FUNCTION "Op20.FCCycles" : VOID	// FC 170
VERSION : 0.1
BEGIN
NETWORK
TITLE =
      A     "OP20".Mode.Automatic;
      FP    "AppoFP_M51.6";
      =     "Op20.Bench.Systems".State.FP_Mode_automatic;
      AN    "OP20".Diagnostic.Alarm_Stop_Cycle;
      AN    "OP20".Diagnostic.Alarm_Emergency;
      FP    "AppoFP_M51.7";
      =     "Op20.Bench.Systems".State.FP_uscita_da_allarme;
NETWORK
TITLE = Attiva ciclo
      A     "Op20.Bench.Systems".State.FP_Mode_automatic;
      O     "Op20.Bench.Systems".State.FP_uscita_da_allarme;
      A(;
      AN    "Op20.Bench.MapE".Index_cassetto_Giu;
      ON    "Op20.Bench.MapE".Gruppo_piantaggio_Su;
      ON    "Op20.Bench.MapE".Piantaggio_Su;
      );
      S     "Op20.Cycles".Restore.Command.Activate_Cycle;
      AN    "OP20".Mode.Automatic;
      O     "OP20".Diagnostic.Alarm_Stop_Cycle;
      O     "OP20".Diagnostic.Alarm_Emergency;
      O     "Op20.Cycles".Restore.State.State_Bit[60];
      R     "Op20.Cycles".Restore.Command.Activate_Cycle;
      CLR;
      =     "OP20".Diagnostic.Hold_State;
      CALL  "Op20.Cycle.Restore" , "OP20.Ist.Cycle.Restore" (
           IN_Cm_ON                 := "Op20.Cycles".Restore.Command.Activate_Cycle,
           IN_HOLD                  := "OP20".Diagnostic.Hold_State,
           IN_STEP                  := FALSE,
           OUT_St_CicloInCorso      := "Op20.Cycles".Restore.State.Cycle_In_Progress,
           OUT_St_CicloTerminatoOK  := "Op20.Cycles".Restore.State.Cycle_Ended_OK,
           OUT_St_CicloTerminatoKO  := "Op20.Cycles".Restore.State.Cycle_Ended_KO,
           OUT_CicloStato           := "Op20.Cycles".Restore.State.State,
           OUT_Page                 := "Op20.Cycles".Restore.State.Page,
           OUT_Message              := "Op20.Cycles".Restore.State.Message);
NETWORK
TITLE = Attiva ciclo
      A     "OP20".Mode.Automatic;
      AN    "OP20".Diagnostic.Alarm_Stop_Cycle;
      AN    "OP20".Diagnostic.Alarm_Emergency;
      AN    "Op20.Cycles".Restore.Command.Activate_Cycle;
// condizione di sicurezza
      =     "Op20.Cycles".General.Command.Activate_Cycle;
      CALL  "Op20.Cycle.General" , "OP20.Ist.Cycle.General" (
           IN_Cm_ON                 := "Op20.Cycles".General.Command.Activate_Cycle,
           IN_HOLD                  := "OP20".Diagnostic.Hold_State,
           IN_STEP                  := FALSE,
           OUT_St_CicloInCorso      := "Op20.Cycles".General.State.Cycle_In_Progress,
           OUT_St_CicloTerminatoOK  := "Op20.Cycles".General.State.Cycle_Ended_OK,
           OUT_St_CicloTerminatoKO  := "Op20.Cycles".General.State.Cycle_Ended_KO,
           OUT_CicloStato           := "Op20.Cycles".General.State.State,
           OUT_Page                 := "Op20.Cycles".General.State.Page,
           OUT_Message              := "Op20.Cycles".General.State.Message);
END_FUNCTION

FUNCTION "OP40.FCMain" : VOID	// FC 200
VERSION : 0.1
VAR_TEMP
  ErrorToolType : BOOL ;
END_VAR
BEGIN
NETWORK
TITLE =
NETWORK
TITLE = OP40 ToolType error
      CALL  "Op40.Bench.FCMapE";
      CALL  "Op40.Tool.FCMapE" (
           ToolType                 := "Op40.Bench.Recipe".ToolType,
           ErrorToolType            := #ErrorToolType);
      A     #ErrorToolType;
      AN    "Op40.Bench.Recipe".Disable.CkCodicePortapezzo;
      S     "Op40.Bench.Alarms".StopCycle.Alarm09;
      CALL  "Op40.Bench.FCConfig";
NETWORK
TITLE =
      A     "Line.Systems".Command.Reset_allarmi;
      =     "Op40.Bench.Systems".Command.Reset_allarmi;
      A     "Line.Systems".Command.TestLampade;
      =     "Op40.Bench.Systems".Command.TestLampade;
      A     "Line.Systems".State.Porte_chiuse;
      =     "Op40.Bench.Systems".State.Porte_chiuse;
      A     "Line.Systems".State.Porte_chiuse_e_bloccate;
      =     "Op40.Bench.Systems".State.Porte_chiuse_e_bloccate;
      CALL  "Bench.Alarms" (
           NumDBallarmi             := "Op40.Bench.Alarms",
           Reset_Allarmi            := "Op40.Bench.Systems".Command.Reset_allarmi,
           AllarmeEmergenza         := "OP40".Diagnostic.Alarm_Emergency,
           AllarmeStopCiclo         := "OP40".Diagnostic.Alarm_Stop_Cycle,
           AllarmeStartCiclo        := "OP40".Diagnostic.Alarm_No_Restart,
           AllarmeWarning           := "OP40".Diagnostic.Alarm_Warning);
      A     "Line".Mode.Emergency;
      =     "OP40".Mode.Emergency;
      A     "Line".Mode.Test_Machine;
      =     "OP40".Mode.Test_Machine;
      A     "Line".Mode.Setup;
      =     "OP40".Mode.Setup;
      A     "Line".Mode.Manual;
      =     "OP40".Mode.Manual;
      A     "Line".Mode.Automatic;
      =     "OP40".Mode.Automatic;
NETWORK
TITLE =
      CALL  "Op40.Bench.FCSystems";
      CALL  "Op40.FCCycles";
NETWORK
TITLE =
      CALL  "Op40.Bench.FCMapA";
END_FUNCTION

FUNCTION "Op40.Bench.FCMapE" : VOID	// FC 201
VERSION : 0.1
BEGIN
NETWORK
TITLE = (start ciclo)
      A     I 6.1;
      =     "Op40.Bench.MapE".PLS_Operator_confirm;
      A     I 9.6;
      =     "Op40.Bench.MapE".Pipe_placed;
      AN    I 9.0;
      =     "Op40.Bench.MapE".Box_out;
      A     I 9.1;
      =     "Op40.Bench.MapE".Box_in;
      A     I 9.2;
      =     "Op40.Bench.MapE".Box_index_up;
      A     I 9.3;
      =     "Op40.Bench.MapE".Box_index_down;
      A     I 9.4;
      =     "Op40.Bench.MapE".Unlock_parts_down;
      A     I 9.5;
      =     "Op40.Bench.MapE".Unlock_parts_up;
      AN    I 1.5;
      =     "Op40.Bench.MapE".PLS_Stop_Cycle;
      A     I 9.7;
      =     "Op40.Bench.MapE".Ring_lock_pipe_present;
END_FUNCTION

FUNCTION "Op40.Bench.FCMapA" : VOID	// FC 202
VERSION : 0.1
BEGIN
NETWORK
TITLE =
      A     "Op40.Bench.MapA".Fine_ciclo_OK;
      =     Q 0.1;
      A     "Op40.Bench.MapA".Fine_ciclo_NON_OK;
      =     Q 0.2;
      A     "Op40.Bench.MapA".EV_abb_index_cassetto;
      =     Q 2.6;
      A     "Op40.Bench.MapA".EV_alza_index_cassetto;
      =     Q 2.7;
      A     "Op40.Bench.MapA".EV_sblocco_pezzo;
      =     Q 3.1;
      A     "Op40.Bench.MapA".EV_blocco_pezzo;
      =     Q 3.0;
END_FUNCTION

FUNCTION "Op40.Bench.FCConfig" : VOID	// FC 203
VERSION : 0.1
BEGIN
NETWORK
TITLE =
END_FUNCTION

FUNCTION "Op40.Bench.FCSystems" : VOID	// FC 205
VERSION : 0.1
VAR_TEMP
  Cmd_abbassa_indc : BOOL ;
  Cmd_alza_indc : BOOL ;
  Cmd_abbassa_indc_ibl : BOOL ;
  Cmd_alza_indc_ibl : BOOL ;
  Cmd_sblocca_pezzo : BOOL ;
  Cmd_blocca_pezzo : BOOL ;
  Cmd_sblocca_pezzo_ibl : BOOL ;
  Cmd_blocca_pezzo_ibl : BOOL ;
  Punt1 : DINT ;
  TempoTime : TIME ;
  TempoS5T : S5TIME ;
  Pos_comandata_asse_X : DINT ;
  Pos_comandata_asse_Y : DINT ;
  Tempo_ribaditura : DINT ;
END_VAR
BEGIN
NETWORK
TITLE = ******************       Diagnostica       *******************
NETWORK
TITLE = Allarmi di emergenza
NETWORK
TITLE = Controllo toolcode 
      L     DB206.DBB 0;
      L     W#16#1F;
      AW;
      L     "Op40.Bench.Recipe".ToolCode;
      <>I;
      AN    "Op40.Bench.Recipe".Disable.CkCodicePortapezzo;
      S     "Op40.Bench.Alarms".StopCycle.Alarm10;
NETWORK
TITLE = Allarmi di STOP CICLO
NETWORK
TITLE = Controllo anelli adattamento
      A     "Op40.Bench.Recipe".Anello1Abilitato;
      AN    "Op40.Tools.MapE".Anello_1_Inserito;
      O(;
      AN    "Op40.Bench.Recipe".Anello1Abilitato;
      A     "Op40.Tools.MapE".Anello_1_Inserito;
      );
      AN    "Op40.Bench.Recipe".Disable.CkPresAnelloAdattamento;
      S     "Op40.Bench.Alarms".StopCycle.Alarm01;
      A     "Op40.Bench.Recipe".Anello2Abilitato;
      AN    "Op40.Tools.MapE".Anello_2_Inserito;
      O(;
      AN    "Op40.Bench.Recipe".Anello2Abilitato;
      A     "Op40.Tools.MapE".Anello_2_Inserito;
      );
      AN    "Op40.Bench.Recipe".Disable.CkPresAnelloAdattamento;
      S     "Op40.Bench.Alarms".StopCycle.Alarm02;
NETWORK
TITLE = Allarmi di NON START CICLO
NETWORK
TITLE = Allarmi di Warning
NETWORK
TITLE = Diagnostica: Hold Macchina
      AN    "OP40".Diagnostic.Alarm_Emergency;
      A(;
      A     "OP40".Mode.Automatic;
      AN    "OP40".Diagnostic.Alarm_Stop_Cycle;
      A     "Op40.Bench.Systems".State.Porte_chiuse_e_bloccate;
      O(;
      A     "OP40".Mode.Manual;
      A     "Op40.Bench.Systems".State.Porte_chiuse;
      );
      );
      =     "OP40".Diagnostic.Safe_State;
NETWORK
TITLE = ******************          Stati            *******************
      A     "Op40.Bench.MapE".Box_out;
      =     "Op40.Bench.Systems".State.Cassetto_fuori;
      A     "Op40.Bench.MapE".Box_in;
      =     "Op40.Bench.Systems".State.Cassetto_dentro;
NETWORK
TITLE =
      A     "Line.Systems".State.Ribaditrice_alta;
      =     "Op40.Bench.Systems".State.Ribaditrice_alta;
      A     "Line.Systems".State.Ribaditrice_bassa;
      =     "Op40.Bench.Systems".State.Ribaditrice_bassa;
      A     "Line.Systems".State.Ribadit_Motore_in_marcia;
      =     "Op40.Bench.Systems".State.Ribaditrice_in_marcia;
      AN    "Line.Systems".State.AsseX_inMovimento;
      AN    "Line.Systems".State.AsseY_inMovimento;
      =     "Op40.Bench.Systems".State.Assi_fermi;
NETWORK
TITLE = Stato: Fronte Start Ciclo
      A     "Op40.Bench.MapE".PLS_Operator_confirm;
      FP    "AppoFP_M50.7";
      =     "Op40.Bench.Systems".Command.FP_Consenso_operatore;
NETWORK
TITLE = Lampade
      A     "Op40.Bench.Systems".State.Ribaditura_pezzo_OK;
      A     "OP40".Mode.Automatic;
      O     "Op40.Bench.Systems".Command.TestLampade;
      =     "Op40.Bench.MapA".Fine_ciclo_OK;
      A     "Op40.Bench.Systems".State.Ribaditura_pezzo_KO;
      A     "OP40".Mode.Automatic;
      O     "Op40.Bench.Systems".Command.TestLampade;
      =     "Op40.Bench.MapA".Fine_ciclo_NON_OK;
NETWORK
TITLE = Cycle Type
NETWORK
TITLE = ******************         Sistemi           *******************
NETWORK
TITLE = Alza/abbassa Index cassetto
//*************************** COMANDI DA CICLI *************************
      A     "Op40.Cycles".General.State.State_Bit[13];
      O     "Op40.Cycles".General.State.State_Bit[35];
      O     "Op40.Cycles".Restore.State.State_Bit[15];
      =     "Op40.Bench.Systems".Command.Abbassa_index_cassetto;
      A     "Op40.Cycles".General.State.State_Bit[16];
      A     "Op40.Bench.Systems".State.Cassetto_dentro;
      O(;
      A     "Op40.Cycles".General.State.State_Bit[40];
      O     "Op40.Cycles".Restore.State.State_Bit[20];
      A     "Op40.Bench.Systems".State.Cassetto_fuori;
      );
      =     "Op40.Bench.Systems".Command.Alza_index_cassetto;
//*************************** COMANDI SENZA INTERBLOCCHI ***************
//CMD---------->Comando abbassa index cassetto
//MANUALE
      A     "Line.OperatorPanel".Commands.Man_40_IndexCassetto;
      A     "Line.MapE".Jog_meno;
      A     "OP40".Mode.Manual;
//AUTOMATICO
      O(;
      A     "OP40".Mode.Automatic;
      AN    "OP40".Diagnostic.Hold_State;
      A     "Op40.Bench.Systems".Command.Abbassa_index_cassetto;
      );
//SICUREZZA
      A     "OP40".Diagnostic.Safe_State;
      =     #Cmd_abbassa_indc;
//CMD---------->Comando alza index cassetto
//MANUALE
      A     "Line.OperatorPanel".Commands.Man_40_IndexCassetto;
      A     "Line.MapE".Jog_piu;
      A     "OP40".Mode.Manual;
//AUTOMATICO
      O(;
      A     "OP40".Mode.Automatic;
      AN    "OP40".Diagnostic.Hold_State;
      A     "Op40.Bench.Systems".Command.Alza_index_cassetto;
      );
//SICUREZZA
      A     "OP40".Diagnostic.Safe_State;
      =     #Cmd_alza_indc;
//************************** INTERBLOCCHI (E SEGNALAZIONE) ****************************
      A     "Op40.Bench.Systems".Command.Reset_allarmi;
      O     "Op40.Bench.Systems".State.Cassetto_dentro;
      O     "Op40.Bench.Systems".State.Cassetto_fuori;
      R     "Op40.Bench.Alarms".Warning.Alarm01;
      A     #Cmd_alza_indc;
      A(;
      AN    "Op40.Bench.Systems".State.Cassetto_dentro;
      AN    "Op40.Bench.Systems".State.Cassetto_fuori;
      );
      S     "Op40.Bench.Alarms".Warning.Alarm01;
// MSG sblocco solo con ribaditrice alta
      A     "Op40.Bench.Systems".Command.Reset_allarmi;
      O     "Op40.Bench.Systems".State.Ribaditrice_alta;
      R     "Op40.Bench.Alarms".Warning.Alarm03;
      A     #Cmd_abbassa_indc;
      AN    "Op40.Bench.Systems".State.Ribaditrice_alta;
      S     "Op40.Bench.Alarms".Warning.Alarm03;
// MSG sblocco solo con assi fermi
      A     "Op40.Bench.Systems".Command.Reset_allarmi;
      O     "Op40.Bench.Systems".State.Assi_fermi;
      R     "Op40.Bench.Alarms".Warning.Alarm04;
      A     #Cmd_abbassa_indc;
      AN    "Op40.Bench.Systems".State.Assi_fermi;
      S     "Op40.Bench.Alarms".Warning.Alarm04;
// MSG sblocco solo con pezzo bloccato
      A     "Op40.Bench.Systems".Command.Reset_allarmi;
      O     "Op40.Bench.Systems".State.Pezzo_bloccato;
      R     "Op40.Bench.Alarms".Warning.Alarm05;
      A     #Cmd_abbassa_indc;
      AN    "Op40.Bench.Systems".State.Pezzo_bloccato;
      S     "Op40.Bench.Alarms".Warning.Alarm05;
//************************** COMANDI CON INTERBLOCCHI ******************************
      AN    "Op40.Bench.Alarms".Warning.Alarm03;
      AN    "Op40.Bench.Alarms".Warning.Alarm04;
      AN    "Op40.Bench.Alarms".Warning.Alarm05;
      A     #Cmd_abbassa_indc;
      =     #Cmd_abbassa_indc_ibl;
      AN    "Op40.Bench.Alarms".Warning.Alarm01;
      A     #Cmd_alza_indc;
      =     #Cmd_alza_indc_ibl;
      CALL  "Std System.Cylinder" , "Ist_cil_40_Index_cass" (
           IN_Enable                := TRUE,
           IN_Command_CylForward    := #Cmd_alza_indc_ibl,
           IN_Command_CylBack       := #Cmd_abbassa_indc_ibl,
           IN_EndStroke_Forward     := "Op40.Bench.MapE".Box_index_down,
           IN_EndStroke_Back        := "Op40.Bench.MapE".Box_index_up,
           IN_Alarms_Reset          := "Op40.Bench.Systems".Command.Reset_allarmi,
           IN_Alarms_TimeOut        := T#3S,
           IN_Hold_Condition        := FALSE,
           OUT_EV_Forward           := "Op40.Bench.MapA".EV_alza_index_cassetto,
           OUT_EV_Back              := "Op40.Bench.MapA".EV_abb_index_cassetto,
           OUT_State_CylForward     := "Op40.Bench.Systems".State.Index_cassetto_alto,
           OUT_State_CylBack        := "Op40.Bench.Systems".State.Index_cassetto_basso,
           OUT_Alarm_ES_Forward     := "Op40.Bench.Alarms".StopCycle.Alarm03,
           OUT_Alarm_ES_Back        := "Op40.Bench.Alarms".StopCycle.Alarm04,
           OUT_Alarm_ForwBack       := "Op40.Bench.Alarms".StopCycle.Alarm05);
NETWORK
TITLE = Blocco/Sblocco pezzo
//*************************** COMANDI DA CICLI *************************
      A     "Op40.Cycles".General.State.State_Bit[10];
      O     "Op40.Cycles".General.State.State_Bit[40];
      O     "Op40.Cycles".Restore.State.State_Bit[20];
      A     "Op40.Bench.MapE".Box_index_down;
      A     "Op40.Bench.Systems".State.Cassetto_fuori;
      =     "Op40.Bench.Systems".Command.Sblocca_pezzo;
      A     "Op40.Cycles".General.State.State_Bit[11];
      O     "Op10.Cycles".General.State.State_Bit[16];
      =     "Op40.Bench.Systems".Command.Blocca_pezzo;
//*************************** COMANDI SENZA INTERBLOCCHI ***************
//CMD---------->Comando sblocco
//MANUALE
      A     "Line.OperatorPanel".Commands.Man_40_BloccoPezzo;
      A     "Line.MapE".Jog_piu;
      A     "OP40".Mode.Manual;
//AUTOMATICO
      O(;
      A     "OP40".Mode.Automatic;
      AN    "OP40".Diagnostic.Hold_State;
      A     "Op40.Bench.Systems".Command.Sblocca_pezzo;
      );
//SICUREZZA
      A     "OP40".Diagnostic.Safe_State;
      =     #Cmd_sblocca_pezzo;
//CMD---------->Comando alza ribaditrice
//MANUALE
      A     "Line.OperatorPanel".Commands.Man_40_BloccoPezzo;
      A     "Line.MapE".Jog_meno;
      A     "OP40".Mode.Manual;
//AUTOMATICO
      O(;
      A     "OP40".Mode.Automatic;
      AN    "OP40".Diagnostic.Hold_State;
      A     "Op40.Bench.Systems".Command.Blocca_pezzo;
      );
//SICUREZZA
      A     "OP40".Diagnostic.Safe_State;
      =     #Cmd_blocca_pezzo;
//************************** INTERBLOCCHI (E SEGNALAZIONE) ****************************
//MSG---> Segnalazione interblocco Movimento ribaditrice non ammesso con motore ribaditrice in marcia
      A     "Op40.Bench.Systems".Command.Reset_allarmi;
      O(;
      A     "Op40.Bench.Systems".State.Cassetto_fuori;
      A     "Op40.Bench.Systems".State.Index_cassetto_alto;
      );
      R     "Op40.Bench.Alarms".Warning.Alarm02;
      A     #Cmd_sblocca_pezzo;
      A(;
      AN    "Op40.Bench.Systems".State.Cassetto_fuori;
      ON    "Op40.Bench.Systems".State.Index_cassetto_alto;
      );
      S     "Op40.Bench.Alarms".Warning.Alarm02;
//************************** COMANDI CON INTERBLOCCHI ******************************
//CMD-------------> Comando abbassa e alza
      AN    "Op40.Bench.Alarms".Warning.Alarm02;
      A     #Cmd_sblocca_pezzo;
      =     #Cmd_sblocca_pezzo_ibl;
      A     #Cmd_blocca_pezzo;
      =     #Cmd_blocca_pezzo_ibl;
      CALL  "Std System.Cylinder" , "Ist_40_CilBloccoPezzo" (
           IN_Enable                := TRUE,
           IN_Command_CylForward    := #Cmd_sblocca_pezzo_ibl,
           IN_Command_CylBack       := #Cmd_blocca_pezzo_ibl,
           IN_EndStroke_Forward     := "Op40.Bench.MapE".Unlock_parts_up,
           IN_EndStroke_Back        := "Op40.Bench.MapE".Unlock_parts_down,
           IN_Alarms_Reset          := "Op40.Bench.Systems".Command.Reset_allarmi,
           IN_Alarms_TimeOut        := T#3S,
           IN_Hold_Condition        := FALSE,
           OUT_EV_Forward           := "Op40.Bench.MapA".EV_sblocco_pezzo,
           OUT_EV_Back              := "Op40.Bench.MapA".EV_blocco_pezzo,
           OUT_State_CylForward     := "Op40.Bench.Systems".State.Pezzo_sbloccato,
           OUT_State_CylBack        := "Op40.Bench.Systems".State.Pezzo_bloccato,
           OUT_Alarm_ES_Forward     := "Op40.Bench.Alarms".StopCycle.Alarm06,
           OUT_Alarm_ES_Back        := "Op40.Bench.Alarms".StopCycle.Alarm07,
           OUT_Alarm_ForwBack       := "Op40.Bench.Alarms".StopCycle.Alarm08);
NETWORK
TITLE = Gestione numero ribaditura in corso
      AN    "Op40.Cycles".General.Command.Activate_Cycle;
      O     "Op40.Cycles".General.State.State_Bit[10];
      O     "Op40.Cycles".General.State.State_Bit[16];
      O     "Op40.Cycles".General.State.State_Bit[40];
      JCN   nAzz;
      L     0;
      T     "Op40.Bench.Systems".Data.Num_punto_in_lavorazione;
nAzz: NOP   0;
      A     "Op40.Cycles".General.State.State_Bit[20];
      FP    "AppoFP_M50.6";
      =     "Op40.Bench.Systems".State.FP_stato_20_generale;
      AN    "Op40.Bench.Systems".State.FP_stato_20_generale;
      JC    nIn;
      L     "Op40.Bench.Systems".Data.Num_punto_in_lavorazione;
      L     1;
      +I;
      T     "Op40.Bench.Systems".Data.Num_punto_in_lavorazione;
nIn:  NOP   0;
NETWORK
TITLE = Valori posizione ribaditura corrente
      L     "Op40.Bench.Systems".Data.Num_punto_in_lavorazione;
      L     0;
      >I;
      JC    Cal;
// Punto inesistente
      L     L#0;
      T     "Op40.Bench.Systems".Data.Pos_comandata_asse_X;
      T     "Op40.Bench.Systems".Data.Pos_comandata_asse_Y;
      T     "Op40.Bench.Systems".Data.Tempo_ribaditura;
      JU    Cen;
Cal:  NOP   0;	// Estrazione dati punto da ricetta
      L     "Op40.Bench.Systems".Data.Num_punto_in_lavorazione;
      DEC   1;
      ITD;
      L     L#12;
      *D;
      L     L#82;
      +D;
      SLW   3;
      T     #Punt1;
      OPN   "Op40.Bench.Recipe";
      L     DBD [#Punt1];
      T     #Pos_comandata_asse_X;
      L     #Punt1;
      L     32;
      +D;
      T     #Punt1;
      L     DBD [#Punt1];
      T     #Pos_comandata_asse_Y;
      L     #Punt1;
      L     32;
      +D;
      T     #Punt1;
      L     DBD [#Punt1];
      T     #Tempo_ribaditura;
      L     #Pos_comandata_asse_X;
      T     "Op40.Bench.Systems".Data.Pos_comandata_asse_X;
      L     #Pos_comandata_asse_Y;
      T     "Op40.Bench.Systems".Data.Pos_comandata_asse_Y;
      L     #Tempo_ribaditura;
      T     "Op40.Bench.Systems".Data.Tempo_ribaditura;
Cen:  NOP   0;
NETWORK
TITLE = Impegno, comandi e stati ribaditrice per lavoro su OP10
      A     "Op40.Cycles".General.State.State_Bit[16];
      O     "Op40.Cycles".General.State.State_Bit[20];
      O     "Op40.Cycles".General.State.State_Bit[25];
      O     "Op40.Cycles".General.State.State_Bit[30];
      A     "Op40.Cycles".General.Command.Activate_Cycle;
      O(;
      A     "Op40.Cycles".Restore.State.State_Bit[10];
      A     "Op40.Cycles".Restore.Command.Activate_Cycle;
      );
      =     "Op40.Bench.Systems".Command.Prenota_ribaditrice;
      A     "Op40.Cycles".General.State.State_Bit[20];
      O     "Op40.Cycles".General.State.State_Bit[25];
      O     "Op40.Cycles".General.State.State_Bit[30];
      =     "Op40.Bench.Systems".Command.Marcia_ribaditrice;
      A     "Op40.Cycles".General.State.State_Bit[25];
      A     "Op40.Bench.Systems".State._Ribaditrice_a_disposiz;
      =     "Op40.Bench.Systems".Command.Abbassa_ribaditrice;
      A     "Op40.Cycles".General.State.State_Bit[13];
      AN    "Op40.Bench.Systems".State._Ribad_in_fuori_ingombro;
      O     "Op40.Cycles".General.State.State_Bit[30];
      O     "Op40.Cycles".Restore.State.State_Bit[10];
      A     "Op40.Bench.Systems".State._Ribaditrice_a_disposiz;
      =     "Op40.Bench.Systems".Command.Alza_ribaditrice;
      A     "Line.Systems".State.Ribad_prenotata_da_OP40;
      =     "Op40.Bench.Systems".State._Ribaditrice_a_disposiz;
NETWORK
TITLE = Ribaditura
      L     "Op40.Bench.Systems".Data.Tempo_ribaditura;
      T     #TempoTime;
      CALL  "TIM_S5TI" (
           $1                       := #TempoTime,
           $2                       := #TempoS5T);
      A     "Op40.Cycles".General.State.State_Bit[25];
      A     "Op40.Bench.Systems".State.Ribaditrice_in_marcia;
      A     "Op40.Bench.Systems".State.Ribaditrice_bassa;
      L     #TempoS5T;
      SD    "Op40_Tempo_di_ribaditura";
      A     "Op40_Tempo_di_ribaditura";
      =     "Op40.Bench.Systems".State.Ribaditura_effettuata;
NETWORK
TITLE = Assi - movimenti per lavorazioni OP10
      A     "Op40.Cycles".General.State.State_Bit[20];
      A     "Line.Systems".State.Ribad_prenotata_da_OP40;
      =     "Op40.Bench.Systems".Command.Vai_in_posizione_assi;
      A     "Line.Systems".State.AsseX_posizioneRaggiunta;
      A     "Line.Systems".State.AsseY_posizioneRaggiunta;
      A     "Line.Systems".State.Ribad_prenotata_da_OP40;
      =     "Op40.Bench.Systems".State._Assi_posiz_raggiunta;
NETWORK
TITLE = Definizione pezzo buono o scarto
      A     "Op40.Cycles".General.State.State_Bit[35];
      S     "Op40.Bench.Systems".State.Ribaditura_pezzo_OK;
      A     "Op40.Bench.MapE".Unlock_parts_up;
      R     "Op40.Bench.Systems".State.Ribaditura_pezzo_OK;
      A     "Op40.Cycles".Restore.Command.Activate_Cycle;
      A     "Op40.Tools.MapE".Presenza_pin_roller;
      AN    "Op40.Bench.Systems".State.Ribaditura_pezzo_OK;
      S     "Op40.Bench.Systems".State.Ribaditura_pezzo_KO;
      A     "Op40.Bench.MapE".Unlock_parts_up;
      R     "Op40.Bench.Systems".State.Ribaditura_pezzo_KO;
END_FUNCTION

FUNCTION "Op40.Tool.FCMapE" : VOID	// FC 206
VERSION : 0.1
VAR_INPUT
  ToolType : INT ;
END_VAR
VAR_OUTPUT
  ErrorToolType : BOOL ;
END_VAR
BEGIN
NETWORK
TITLE = Tool 1 - mappa ingressi
      L     #ToolType;
      L     1;
      <>I;
      JC    no1;
      SET;
      R     #ErrorToolType;
// Tool 1 - mappa ingressi
      A     I 7.0;
      =     "Op40.Tools.MapE".ToolCode_Bit_0;
      A     I 7.1;
      =     "Op40.Tools.MapE".ToolCode_Bit_1;
      A     I 7.2;
      =     "Op40.Tools.MapE".ToolCode_Bit_2;
      A     I 7.3;
      =     "Op40.Tools.MapE".ToolCode_Bit_3;
      A     I 7.4;
      =     "Op40.Tools.MapE".ToolCode_Bit_4;
      A     I 5.1;
      =     "Op40.Tools.MapE".Anello_1_Inserito;
      A     I 5.2;
      =     "Op40.Tools.MapE".Anello_2_Inserito;
      A     I 5.0;
      =     "Op40.Tools.MapE".Presenza_pin_roller;
      BEU;
no1:  NOP   0;
NETWORK
TITLE = Tool 2 - mappa ingressi
      L     #ToolType;
      L     2;
      <>I;
      JC    no2;
      SET;
      S     #ErrorToolType;
// Tool 2 - predisposto ma inesistente
      BEU;
no2:  NOP   0;
NETWORK
TITLE = Error Tool Type
      SET;
      S     #ErrorToolType;
END_FUNCTION

FUNCTION "Op40.FCCycles" : VOID	// FC 220
VERSION : 0.1
BEGIN
NETWORK
TITLE =
      A     "OP40".Mode.Automatic;
      FP    "AppoFP_M51.0";
      =     "Op40.Bench.Systems".State.FP_Mode_automatic;
      AN    "OP40".Diagnostic.Alarm_Stop_Cycle;
      AN    "OP40".Diagnostic.Alarm_Emergency;
      FP    "AppoFP_M51.1";
      =     "Op40.Bench.Systems".State.FP_uscita_da_allarme;
NETWORK
TITLE =
      A     "Op40.Bench.Systems".State.FP_Mode_automatic;
      O     "Op40.Bench.Systems".State.FP_uscita_da_allarme;
      A(;
      AN    "Op40.Bench.Systems".State.Cassetto_fuori;
      ON    "Op40.Bench.MapE".Box_index_down;
      ON    "Op40.Bench.MapE".Unlock_parts_up;
      );
      S     "Op40.Cycles".Restore.Command.Activate_Cycle;
      AN    "OP40".Mode.Automatic;
      O     "OP40".Diagnostic.Alarm_Stop_Cycle;
      O     "OP40".Diagnostic.Alarm_Emergency;
      O     "Op40.Bench.MapE".PLS_Stop_Cycle;
      O     "Op40.Cycles".Restore.State.State_Bit[60];
      R     "Op40.Cycles".Restore.Command.Activate_Cycle;
      CLR;
      =     "OP40".Diagnostic.Hold_State;
      CALL  "Op40.Cycle.Restore" , "OP40.Ist.Cycle.Restore" (
           IN_Cm_ON                 := "Op40.Cycles".Restore.Command.Activate_Cycle,
           IN_HOLD                  := "OP40".Diagnostic.Hold_State,
           IN_STEP                  := FALSE,
           OUT_St_CicloInCorso      := "Op40.Cycles".Restore.State.Cycle_In_Progress,
           OUT_St_CicloTerminatoOK  := "Op40.Cycles".Restore.State.Cycle_Ended_OK,
           OUT_St_CicloTerminatoKO  := "Op40.Cycles".Restore.State.Cycle_Ended_KO,
           OUT_CicloStato           := "Op40.Cycles".Restore.State.State,
           OUT_Page                 := "Op40.Cycles".Restore.State.Page,
           OUT_Message              := "Op40.Cycles".Restore.State.Message);
NETWORK
TITLE = Attiva ciclo
      A     "OP40".Mode.Automatic;
      AN    "OP40".Diagnostic.Alarm_Stop_Cycle;
      AN    "OP40".Diagnostic.Alarm_Emergency;
      AN    "Op40.Cycles".Restore.Command.Activate_Cycle;
// condizione di sicurezza
      AN    "Op40.Bench.MapE".PLS_Stop_Cycle;
      =     "Op40.Cycles".General.Command.Activate_Cycle;
      CALL  "Op40.Cycle.General" , "OP40.Ist.Cycle.General" (
           IN_Cm_ON                 := "Op40.Cycles".General.Command.Activate_Cycle,
           IN_HOLD                  := "OP40".Diagnostic.Hold_State,
           IN_STEP                  := FALSE,
           OUT_St_CicloInCorso      := "Op40.Cycles".General.State.Cycle_In_Progress,
           OUT_St_CicloTerminatoOK  := "Op40.Cycles".General.State.Cycle_Ended_OK,
           OUT_St_CicloTerminatoKO  := "Op40.Cycles".General.State.Cycle_Ended_KO,
           OUT_CicloStato           := "Op40.Cycles".General.State.State,
           OUT_Page                 := "Op40.Cycles".General.State.Page,
           OUT_Message              := "Op40.Cycles".General.State.Message);
END_FUNCTION

DATA_BLOCK "Line"	// DB 50
VERSION : 0.1
  STRUCT
   Mode : STRUCT
    Emergency : BOOL ;	//MODO Macchina spenta
    Test_Machine : BOOL ;	//MODO Aspetta pressione nel circuito pneumatico e/o idraulico + MODO Test Lampad
    Setup : BOOL ;	//MODO Cambio Ricetta o setup
    Manual : BOOL ;	//MODO Manuale
    Automatic : BOOL ;	//MODO Automatico
    Service : BOOL ;	//MODO Messa in servizio
    Free_06 : BOOL ;
    Free_07 : BOOL ;
   END_STRUCT ;
   Diagnostic : STRUCT
    Alarm_Emergency : BOOL ;	//Macchina in Emergenza
    Alarm_Stop_Cycle : BOOL ;	//Allarme che blocca il ciclo attivo
    Alarm_No_Restart : BOOL ;	//Allarme che blocca un nuovo ciclo
    Alarm_Warning : BOOL ;	//Segnalazione o avvertenza
    Safe_State : BOOL ;	//MODO Sicuro : e' possibile eseguire i comandi manuali in sicurezza
    Initial_Conditions : BOOL ;	//condizioni iniziali macchina
    Hold_State : BOOL ;	//Hold Macchina
    Free_07 : BOOL ;
    ResetAlarm : BOOL ;
   END_STRUCT ;
   Software : STRUCT
    SwName : STRING  [20 ];
    SwVersion : STRING  [11 ];
   END_STRUCT ;
  END_STRUCT ;	
BEGIN
END_DATA_BLOCK

DATA_BLOCK "Line.MapE"	// DB 51
VERSION : 0.1
  STRUCT
   Q_Ribaditrice : BOOL ;
   Q_protezione_uscite : BOOL ;
   Q_Protez_circ_emergena : BOOL ;	//161QF1
   Q_Automatici_230_V : BOOL ;	//162F1-162F2-162F3-162F4
   Aux_OK : BOOL ;
   Ripari_OK : BOOL ;
   Anomalia_Condizionatore : BOOL ;
   Sequenza_fasi_OK : BOOL ;
   PLC_OK : BOOL ;	//Feedback relè PLC ok
   Chiave_Blocc_Porta_SX : BOOL ;
   Chiave_Blocc_Porta_DX : BOOL ;
   P_TestLampade : BOOL ;
   P_StartCiclo : BOOL ;	//??? che fa ???
   P_StopCiclo : BOOL ;
   S_Manuale : BOOL ;
   S_Automatico : BOOL ;
   Q_Azionam_Asse_X : BOOL ;
   Q_Azionam_Asse_Y : BOOL ;
   Jog_piu : BOOL ;
   Jog_meno : BOOL ;
   P_reset_allarmi : BOOL ;
   Pressostato_aria : BOOL ;
   Ribaditrice_bassa : BOOL ;
   Ribaditrice_alta : BOOL ;
   Press_aria_dpoop_EMG : BOOL ;
   Extracorsa_X : BOOL ;
   Extracorsa_Y : BOOL ;
   Ris_33 : BOOL ;
   Ris_34 : BOOL ;
   Ris_35 : BOOL ;
   Ris_36 : BOOL ;
   Ris_37 : BOOL ;
  END_STRUCT ;	
BEGIN
END_DATA_BLOCK

DATA_BLOCK "Line.MapA"	// DB 52
VERSION : 0.1
  STRUCT
   PLC_OK : BOOL ;
   Valvola_generale_aria : BOOL ;	//TOLTO!!!
   Marcia_ribaditrice : BOOL ;
   EV_abbassa_ribaditrice : BOOL ;
   Spare_0_4 : BOOL ;
   Blocco_porta_SX : BOOL ;
   Blocco_porta_DX : BOOL ;
   Lampeggiante_allarmi : BOOL ;
   LampPorteChiuse : BOOL ;
  END_STRUCT ;	
BEGIN
END_DATA_BLOCK

DATA_BLOCK "Line.Config"	// DB 53
VERSION : 0.1
  STRUCT
   Vel_max_assi_auto : DINT ;	//
   Vel_max_assi_man : DINT ;
   Accel_assi_auto : DINT ;
   Accel_assi_man : DINT ;
   Offset_attrezzo_OP10_X : DINT ;	//
   Offset_attrezzo_OP10_Y : DINT ;
   Offset_attrezzo_OP40_X : DINT ;	//
   Offset_attrezzo_OP40_Y : DINT ;
  END_STRUCT ;	
BEGIN
END_DATA_BLOCK

DATA_BLOCK "Line.Alarms"	// DB 54
VERSION : 0.1
  STRUCT
   Emegency : STRUCT
    Alarm01 : BOOL ;	//Q_protezione_uscite
    Alarm02 : BOOL ;	//Protez_circ_emergena
    Alarm03 : BOOL ;	//Sequenza_fasi_OK
    Alarm04 : BOOL ;	//Q_Azionam_Asse_X
    Alarm05 : BOOL ;	//Q_Azionam_Asse_Y
    Alarm06 : BOOL ;	//Manca aria
    Alarm07 : BOOL ;	//Valvola aria inceppata
    Alarm08 : BOOL ;	//Errore comunicazione con Azionamento asse X
    Alarm09 : BOOL ;	//Errore comunicazione con Azionamento asse Y
    Alarm10 : BOOL ;	//Errore comunicazione con CU Azionamento asse X
    Alarm11 : BOOL ;	//Errore comunicazione con CU Azionamento asse Y
    Alarm12 : BOOL ;	//Extracorsa asse X
    Alarm13 : BOOL ;	//Extracorsa asse Y
    Alarm14 : BOOL ;	//Errore Relè PLC OK
    Alarm15 : BOOL ;
    Alarm16 : BOOL ;
    Alarm17 : BOOL ;
    Alarm18 : BOOL ;
    Alarm19 : BOOL ;
    Alarm20 : BOOL ;
    Alarm21 : BOOL ;
    Alarm22 : BOOL ;
    Alarm23 : BOOL ;
    Alarm24 : BOOL ;
    Alarm25 : BOOL ;
    Alarm26 : BOOL ;
    Alarm27 : BOOL ;
    Alarm28 : BOOL ;
    Alarm29 : BOOL ;
    Alarm30 : BOOL ;
    Alarm31 : BOOL ;
    Alarm32 : BOOL ;
    Alarm33 : BOOL ;
    Alarm34 : BOOL ;
    Alarm35 : BOOL ;
    Alarm36 : BOOL ;
    Alarm37 : BOOL ;
    Alarm38 : BOOL ;
    Alarm39 : BOOL ;
    Alarm40 : BOOL ;
    Alarm41 : BOOL ;
    Alarm42 : BOOL ;
    Alarm43 : BOOL ;
    Alarm44 : BOOL ;
    Alarm45 : BOOL ;
    Alarm46 : BOOL ;
    Alarm47 : BOOL ;
    Alarm48 : BOOL ;
    Alarm49 : BOOL ;
    Alarm50 : BOOL ;
    Alarm51 : BOOL ;
    Alarm52 : BOOL ;
    Alarm53 : BOOL ;
    Alarm54 : BOOL ;
    Alarm55 : BOOL ;
    Alarm56 : BOOL ;
    Alarm57 : BOOL ;
    Alarm58 : BOOL ;
    Alarm59 : BOOL ;
    Alarm60 : BOOL ;
    Alarm61 : BOOL ;
    Alarm62 : BOOL ;
    Alarm63 : BOOL ;
    Alarm64 : BOOL ;
   END_STRUCT ;
   StopCycle : STRUCT
    Alarm01 : BOOL ;	//Ribaditrice non bassa
    Alarm02 : BOOL ;	//Ribaditrice non alta
    Alarm03 : BOOL ;	//Incongruenza sensori ribaditrice
    Alarm04 : BOOL ;	//Porte non chiuse
    Alarm05 : BOOL ;	//Chiave non Bloccata Porta SX
    Alarm06 : BOOL ;	//Chiave non Bloccata Porta DX
    Alarm07 : BOOL ;	//asse X bloccato con Ribaditrice non alta
    Alarm08 : BOOL ;	//asse Y bloccato con Ribaditrice non alta
    Alarm09 : BOOL ;
    Alarm10 : BOOL ;
    Alarm11 : BOOL ;	//Macchina in emergenza
    Alarm12 : BOOL ;
    Alarm13 : BOOL ;
    Alarm14 : BOOL ;
    Alarm15 : BOOL ;
    Alarm16 : BOOL ;
    Alarm17 : BOOL ;
    Alarm18 : BOOL ;
    Alarm19 : BOOL ;
    Alarm20 : BOOL ;
    Alarm21 : BOOL ;
    Alarm22 : BOOL ;
    Alarm23 : BOOL ;
    Alarm24 : BOOL ;
    Alarm25 : BOOL ;
    Alarm26 : BOOL ;
    Alarm27 : BOOL ;
    Alarm28 : BOOL ;
    Alarm29 : BOOL ;
    Alarm30 : BOOL ;
    Alarm31 : BOOL ;
    Alarm32 : BOOL ;
    Alarm33 : BOOL ;
    Alarm34 : BOOL ;
    Alarm35 : BOOL ;
    Alarm36 : BOOL ;
    Alarm37 : BOOL ;
    Alarm38 : BOOL ;
    Alarm39 : BOOL ;
    Alarm40 : BOOL ;
    Alarm41 : BOOL ;
    Alarm42 : BOOL ;
    Alarm43 : BOOL ;
    Alarm44 : BOOL ;
    Alarm45 : BOOL ;
    Alarm46 : BOOL ;
    Alarm47 : BOOL ;
    Alarm48 : BOOL ;
    Alarm49 : BOOL ;
    Alarm50 : BOOL ;
    Alarm51 : BOOL ;
    Alarm52 : BOOL ;
    Alarm53 : BOOL ;
    Alarm54 : BOOL ;
    Alarm55 : BOOL ;
    Alarm56 : BOOL ;
    Alarm57 : BOOL ;
    Alarm58 : BOOL ;
    Alarm59 : BOOL ;
    Alarm60 : BOOL ;
    Alarm61 : BOOL ;
    Alarm62 : BOOL ;
    Alarm63 : BOOL ;
    Alarm64 : BOOL ;
   END_STRUCT ;
   RestartCycle : STRUCT
    Alarm01 : BOOL ;
    Alarm02 : BOOL ;
    Alarm03 : BOOL ;
    Alarm04 : BOOL ;
    Alarm05 : BOOL ;
    Alarm06 : BOOL ;
    Alarm07 : BOOL ;
    Alarm08 : BOOL ;
    Alarm09 : BOOL ;
    Alarm10 : BOOL ;
    Alarm11 : BOOL ;
    Alarm12 : BOOL ;
    Alarm13 : BOOL ;
    Alarm14 : BOOL ;
    Alarm15 : BOOL ;
    Alarm16 : BOOL ;
    Alarm17 : BOOL ;
    Alarm18 : BOOL ;
    Alarm19 : BOOL ;
    Alarm20 : BOOL ;
    Alarm21 : BOOL ;
    Alarm22 : BOOL ;
    Alarm23 : BOOL ;
    Alarm24 : BOOL ;
    Alarm25 : BOOL ;
    Alarm26 : BOOL ;
    Alarm27 : BOOL ;
    Alarm28 : BOOL ;
    Alarm29 : BOOL ;
    Alarm30 : BOOL ;
    Alarm31 : BOOL ;
    Alarm32 : BOOL ;
    Alarm33 : BOOL ;
    Alarm34 : BOOL ;
    Alarm35 : BOOL ;
    Alarm36 : BOOL ;
    Alarm37 : BOOL ;
    Alarm38 : BOOL ;
    Alarm39 : BOOL ;
    Alarm40 : BOOL ;
    Alarm41 : BOOL ;
    Alarm42 : BOOL ;
    Alarm43 : BOOL ;
    Alarm44 : BOOL ;
    Alarm45 : BOOL ;
    Alarm46 : BOOL ;
    Alarm47 : BOOL ;
    Alarm48 : BOOL ;
    Alarm49 : BOOL ;
    Alarm50 : BOOL ;
    Alarm51 : BOOL ;
    Alarm52 : BOOL ;
    Alarm53 : BOOL ;
    Alarm54 : BOOL ;
    Alarm55 : BOOL ;
    Alarm56 : BOOL ;
    Alarm57 : BOOL ;
    Alarm58 : BOOL ;
    Alarm59 : BOOL ;
    Alarm60 : BOOL ;
    Alarm61 : BOOL ;
    Alarm62 : BOOL ;
    Alarm63 : BOOL ;
    Alarm64 : BOOL ;
   END_STRUCT ;
   Warning : STRUCT
    Alarm01 : BOOL ;	//Q_Ribaditrice
    Alarm02 : BOOL ;	//Q_Automatici_230_V
    Alarm03 : BOOL ;	//Anomalia_Condizionatore
    Alarm04 : BOOL ;	//Ribaditrice bloccata con motore ribaditrice ferma
    Alarm05 : BOOL ;	//Marcia ribaditrice solo con cassetti OP10 e OP40 indexati
    Alarm06 : BOOL ;	//Dicesa dibaditrice solo con cassetti OP10 e OP40 indexati
    Alarm07 : BOOL ;	//Marcia assi solo con cassetti OP10 e OP40 indexati
    Alarm08 : BOOL ;
    Alarm09 : BOOL ;
    Alarm10 : BOOL ;
    Alarm11 : BOOL ;
    Alarm12 : BOOL ;
    Alarm13 : BOOL ;
    Alarm14 : BOOL ;
    Alarm15 : BOOL ;
    Alarm16 : BOOL ;
    Alarm17 : BOOL ;
    Alarm18 : BOOL ;
    Alarm19 : BOOL ;
    Alarm20 : BOOL ;
    Alarm21 : BOOL ;
    Alarm22 : BOOL ;
    Alarm23 : BOOL ;
    Alarm24 : BOOL ;
    Alarm25 : BOOL ;
    Alarm26 : BOOL ;
    Alarm27 : BOOL ;
    Alarm28 : BOOL ;
    Alarm29 : BOOL ;
    Alarm30 : BOOL ;
    Alarm31 : BOOL ;
    Alarm32 : BOOL ;
    Alarm33 : BOOL ;
    Alarm34 : BOOL ;
    Alarm35 : BOOL ;
    Alarm36 : BOOL ;
    Alarm37 : BOOL ;
    Alarm38 : BOOL ;
    Alarm39 : BOOL ;
    Alarm40 : BOOL ;
    Alarm41 : BOOL ;
    Alarm42 : BOOL ;
    Alarm43 : BOOL ;
    Alarm44 : BOOL ;
    Alarm45 : BOOL ;
    Alarm46 : BOOL ;
    Alarm47 : BOOL ;
    Alarm48 : BOOL ;
    Alarm49 : BOOL ;
    Alarm50 : BOOL ;
    Alarm51 : BOOL ;
    Alarm52 : BOOL ;
    Alarm53 : BOOL ;
    Alarm54 : BOOL ;
    Alarm55 : BOOL ;
    Alarm56 : BOOL ;
    Alarm57 : BOOL ;
    Alarm58 : BOOL ;
    Alarm59 : BOOL ;
    Alarm60 : BOOL ;
    Alarm61 : BOOL ;
    Alarm62 : BOOL ;
    Alarm63 : BOOL ;
    Alarm64 : BOOL ;
   END_STRUCT ;
  END_STRUCT ;	
BEGIN
END_DATA_BLOCK

DATA_BLOCK "Line.Systems"	// DB 55
VERSION : 0.1
  STRUCT
   Command : STRUCT 	//
    Reset_allarmi : BOOL ;
    TestLampade : BOOL ;	//da programmare sul pannello operatore
    Abbassa_ribaditrice : BOOL ;
    Alza_ribaditrice : BOOL ;
    Marcia_ribaditrice : BOOL ;	//manca ingresso
    Marcia_manuale_ribaditr : BOOL ;
    Posiziona_Assi : BOOL ;
    ris_0_7 : BOOL ;
    AsseX_Enable : BOOL ;
    AsseX_StartPosizionam : BOOL ;
    AsseX_ris_2 : BOOL ;
    AsseX_ris_3 : BOOL ;
    AsseX_ris_4 : BOOL ;
    AsseX_ris_5 : BOOL ;
    AsseX_ris_6 : BOOL ;
    AsseX_ris_7 : BOOL ;
    AsseY_Enable : BOOL ;
    AsseY_StartPosizionam : BOOL ;
    AsseY_ris_2 : BOOL ;
    AsseY_ris_3 : BOOL ;
    AsseY_ris_4 : BOOL ;
    AsseY_ris_5 : BOOL ;
    AsseY_ris_6 : BOOL ;
    AsseY_ris_7 : BOOL ;
    PrenotaRib_OP10 : BOOL ;
    PrenotaRib_OP40 : BOOL ;
    ris_w4 : WORD ;
    ris_w6 : DWORD ;
   END_STRUCT ;
   State : STRUCT 	//da ind. 10
    PLC_OK : BOOL ;
    Porte_chiuse : BOOL ;
    Ribadit_Motore_in_marcia : BOOL ;
    Ribaditrice_bassa : BOOL ;
    Ribaditrice_alta : BOOL ;
    Porte_chiuse_e_bloccate : BOOL ;
    Cassetto_OP10_indexato : BOOL ;
    Cassetto_OP40_indexato : BOOL ;
    AsseX_referenziato : BOOL ;
    AsseX_posizioneRaggiunta : BOOL ;
    AsseX_inMovimento : BOOL ;
    Ris_1_3 : BOOL ;
    AsseX_ExtracorsaOK : BOOL ;
    AsseX_FC_indietro : BOOL ;
    AsseX_FC_avanti : BOOL ;
    AsseX_Pronto : BOOL ;
    AsseY_referenziato : BOOL ;
    AsseY_posizioneRaggiunta : BOOL ;
    AsseY_inMovimento : BOOL ;
    Ris_2_3 : BOOL ;
    AsseY_ExtracorsaOK : BOOL ;
    AsseY_FC_indietro : BOOL ;
    AsseY_FC_avanti : BOOL ;
    AsseY_pronto : BOOL ;
    Ribad_prenotata_da_OP10 : BOOL ;
    Ribad_prenotata_da_OP40 : BOOL ;
    FP_IngressoInPag_TeachIn : BOOL ;
    FP_NumPuntoCambiato : BOOL ;
    FP_RichiestaLeggiPunto : BOOL ;
    FP_RichiestaSalvaPunto : BOOL ;
    FP_RichiestaTeachInPunto : BOOL ;
    ris_w4 : WORD ;
    ris_w6 : DWORD ;
   END_STRUCT ;
   Data : STRUCT 	//da ind. 20
    ris_X_0 : INT ;
    AsseX_Accelerazione : INT ;
    AsseX_Decellerazione : INT ;
    AsseX_Velocita : DINT ;
    AsseX_PosizioneComandata : DINT ;
    AsseX_PosizioneAttuale : DINT ;
    AsseX_CodiceErrore : BYTE ;
    AsseX_ris20 : WORD ;
    AsseX_ris22 : DWORD ;
    AsseX_ris26 : DWORD ;
    ris_Y_30 : INT ;
    AsseY_Accelerazione : INT ;
    AsseY_Decellerazione : INT ;
    AsseY_Velocita : DINT ;
    AsseY_PosizioneComandata : DINT ;
    AsseY_PosizioneAttuale : DINT ;
    AsseY_CodiceErrore : BYTE ;
    AsseY_ris50 : WORD ;
    AsseY_ris52 : DWORD ;
    AsseY_ris56 : DWORD ;
    PuntoInTeachIn : INT ;
    ris_82 : INT ;
    ris_84 : INT ;
    ris_86 : DINT ;
    ris_90 : ARRAY  [0 .. 40 ] OF INT ;
   END_STRUCT ;
  END_STRUCT ;	
BEGIN
END_DATA_BLOCK

DATA_BLOCK "Line.Cycles"	// DB 60
VERSION : 0.1
  STRUCT
   Coord_Ribaditrice : UDT 200;
  END_STRUCT ;	
BEGIN
END_DATA_BLOCK

DATA_BLOCK "Line.OperatorPanel"	// DB 70
VERSION : 0.1
  STRUCT
   OP_System_Data : STRUCT
    PageDisplayed : INT ;
    Year_Byte0 : BYTE ;
    Year_Byte1 : BYTE ;
    Month_byte0 : BYTE ;
    Month_byte1 : BYTE ;
    Day_byte0 : BYTE ;
    Day_byte1 : BYTE ;
    HH : BYTE ;
    MM : BYTE ;
    NewPage : INT ;
   END_STRUCT ;
   Commands : STRUCT 	//da indirizzo 12
    Man_Alza_Abb_Ribaditrice : BOOL ;
    Man_Marcia_Ribaditrice : BOOL ;
    Man_Jog_AsseX : BOOL ;
    Man_Jog_AsseY : BOOL ;
    Man_10_IndexCassetto : BOOL ;
    Man_10_BloccoPezzo : BOOL ;
    Man_20_IndexCassetto : BOOL ;
    Man_20_GruppoPiantaggio : BOOL ;
    Man_20_Piantaggio : BOOL ;
    Man_40_IndexCassetto : BOOL ;
    Man_40_BloccoPezzo : BOOL ;
    Man_disp_2_3 : BOOL ;
    Man_disp_2_4 : BOOL ;
    Man_disp_2_5 : BOOL ;
    Man_disp_2_6 : BOOL ;
    Man_disp_2_7 : BOOL ;
    Man_VaiAlPunto : WORD ;
    Reset_Allarmi : BOOL ;
    Cmd_VaiAlPunto : BOOL ;
    Cmd_TeachInPunto : BOOL ;
    Cmd_SalvaPunto : BOOL ;
    Cmd_LeggiPunto : BOOL ;
    Ris_16_5 : BOOL ;
    ris_w18 : DINT ;
    ris_w22 : DINT ;
   END_STRUCT ;
   States : STRUCT 	//da indirizzo 26
    RibaditriceAlta : BOOL ;
    RibaditriceBassa : BOOL ;
    RibaditriceFerma : BOOL ;
    RibaditriceInMarcia : BOOL ;
    OP10IndexCassSbloccato : BOOL ;
    OP10IndexCassBloccato : BOOL ;
    OP10PezzoSbloccato : BOOL ;
    OP10PezzoBloccato : BOOL ;
    AsseXIndietro : BOOL ;
    AsseXAvanti : BOOL ;
    AsseYIndietro : BOOL ;
    AsseYAvanti : BOOL ;
    OP20IndexCassSbloccato : BOOL ;
    OP20IndexCassBloccato : BOOL ;
    OP20GrPiantaggioAlto : BOOL ;
    OP20GrPiantaggioBasso : BOOL ;
    OP20PiantaggioAlto : BOOL ;
    OP20PiantaggioBasso : BOOL ;
    OP40IndexCassSbloccato : BOOL ;
    OP40IndexCassBloccato : BOOL ;
    OP40PezzoSbloccato : BOOL ;
    OP40PezzoBloccato : BOOL ;
    Op10_recipe : BOOL ;
    Op20_recipe : BOOL ;
    Op40_recipe : BOOL ;
    ris_B31 : BYTE ;
    ris_w32 : DINT ;
   END_STRUCT ;
   Data : STRUCT 	//da indirizzo 36
    AsseX_PosizioneAttuale : DINT ;	//Valori assoluti assi
    AsseY_PosizioneAttuale : DINT ;	//Valori assoluti assi
    PosizionePunzone : REAL ;
    Cmd_Override_man : INT ;
    Cmd_Override_auto : INT ;
    AsseX_PosAttualeOP10 : DINT ;
    AsseY_PosAttualeOP10 : DINT ;
    AsseX_PosAttualeOP40 : DINT ;
    AsseY_PosAttualeOP40 : DINT ;
    Cmd_PuntoSelezionato : INT ;
    Min_PerSelezionePunto : INT ;
    Max_PerSelezionePunto : INT ;
    X_PosPuntoSelezionato : DINT ;
    Y_PosPuntoSelezionato : DINT ;
    TempoRibad_PuntoSelez : DINT ;
    ris_array : ARRAY  [0 .. 15 ] OF REAL ;
   END_STRUCT ;
   cycles : STRUCT 	//indirizzo 150
    OP10_cycle_general : BOOL ;
    OP10_cycle_restore : BOOL ;
    OP20_cycle_general : BOOL ;
    OP20_cycle_restore : BOOL ;
    OP40_cycle_general : BOOL ;
    OP40_cycle_restore : BOOL ;
    OP10_message : INT ;
    OP10_spacer : INT ;
    OP40_message : INT ;
    OP40_spacer : INT ;
    OP20_message : INT ;
    Line_State : INT ;
    ris_w8 : INT ;
    ris_array : ARRAY  [0 .. 16 ] OF INT ;
   END_STRUCT ;
  END_STRUCT ;	
BEGIN
END_DATA_BLOCK

DATA_BLOCK "OP10"	// DB 100
VERSION : 0.1
  STRUCT
   Mode : STRUCT
    Emergency : BOOL ;	//MODO Macchina spenta
    Test_Machine : BOOL ;	//MODO Aspetta pressione nel circuito pneumatico e/o idraulico + MODO Test Lampad
    Setup : BOOL ;	//MODO Cambio Ricetta o setup
    Manual : BOOL ;	//MODO Manuale
    Automatic : BOOL ;	//MODO Automatico
    Service : BOOL ;	//MODO Messa in servizio
    Free_06 : BOOL ;
    Free_07 : BOOL ;
   END_STRUCT ;
   Diagnostic : STRUCT
    Alarm_Emergency : BOOL ;	//Macchina in Emergenza
    Alarm_Stop_Cycle : BOOL ;	//Allarme che blocca il ciclo attivo
    Alarm_No_Restart : BOOL ;	//Allarme che blocca un nuovo ciclo
    Alarm_Warning : BOOL ;	//Segnalazione o avvertenza
    Safe_State : BOOL ;	//MODO Sicuro : e' possibile eseguire i comandi manuali in sicurezza
    Initial_Conditions : BOOL ;	//condizioni iniziali macchina
    Hold_State : BOOL ;	//Hold Macchina
    Free_07 : BOOL ;
    ResetAlarm : BOOL ;
   END_STRUCT ;
   Software : STRUCT
    SwName : STRING  [20 ];
    SwVersion : STRING  [11 ];
   END_STRUCT ;
  END_STRUCT ;	
BEGIN
END_DATA_BLOCK

DATA_BLOCK "Op10.Bench.MapE"	// DB 101
VERSION : 0.1
  STRUCT
   P_Consenso_operatore : BOOL ;	//(start ciclo)
   Cassetto_fuori : BOOL ;
   Cassetto_dentro : BOOL ;
   Index_cassetto_Giu : BOOL ;
   Index_cassetto_Su : BOOL ;
   Sblocco_pezzo_Giu : BOOL ;
   Sblocco_pezzo_Su : BOOL ;
   PulStopCiclo : BOOL ;
  END_STRUCT ;	
BEGIN
END_DATA_BLOCK

DATA_BLOCK "Op10.Bench.MapA"	// DB 102
VERSION : 0.1
  STRUCT
   Fine_ciclo_OK : BOOL ;	//
   Fine_ciclo_NON_OK : BOOL ;
   EV_abb_index_cassetto : BOOL ;
   EV_alza_index_cassetto : BOOL ;
   EV_sblocco_pezzo : BOOL ;
   EV_blocco_pezzo : BOOL ;	//??? esiste?
  END_STRUCT ;	
BEGIN
END_DATA_BLOCK

DATA_BLOCK "Op10.Bench.Config"	// DB 103
VERSION : 0.1
  STRUCT
   dummy : INT ;
  END_STRUCT ;	
BEGIN
END_DATA_BLOCK

DATA_BLOCK "Op10.Bench.Alarms"	// DB 104
VERSION : 0.1
  STRUCT
   Emegency : STRUCT
    Alarm01 : BOOL ;	//OP10 ToolType error
    Alarm02 : BOOL ;	//OP10 ToolCode error
    Alarm03 : BOOL ;
    Alarm04 : BOOL ;
    Alarm05 : BOOL ;
    Alarm06 : BOOL ;
    Alarm07 : BOOL ;
    Alarm08 : BOOL ;
    Alarm09 : BOOL ;	//
    Alarm10 : BOOL ;	//
    Alarm11 : BOOL ;	//
    Alarm12 : BOOL ;	//
    Alarm13 : BOOL ;	//
    Alarm14 : BOOL ;	//
    Alarm15 : BOOL ;
    Alarm16 : BOOL ;
    Alarm17 : BOOL ;
    Alarm18 : BOOL ;
    Alarm19 : BOOL ;
    Alarm20 : BOOL ;
    Alarm21 : BOOL ;
    Alarm22 : BOOL ;
    Alarm23 : BOOL ;
    Alarm24 : BOOL ;
    Alarm25 : BOOL ;
    Alarm26 : BOOL ;
    Alarm27 : BOOL ;
    Alarm28 : BOOL ;
    Alarm29 : BOOL ;
    Alarm30 : BOOL ;
    Alarm31 : BOOL ;
    Alarm32 : BOOL ;
    Alarm33 : BOOL ;
    Alarm34 : BOOL ;
    Alarm35 : BOOL ;
    Alarm36 : BOOL ;
    Alarm37 : BOOL ;
    Alarm38 : BOOL ;
    Alarm39 : BOOL ;
    Alarm40 : BOOL ;
    Alarm41 : BOOL ;
    Alarm42 : BOOL ;
    Alarm43 : BOOL ;
    Alarm44 : BOOL ;
    Alarm45 : BOOL ;
    Alarm46 : BOOL ;
    Alarm47 : BOOL ;
    Alarm48 : BOOL ;
    Alarm49 : BOOL ;
    Alarm50 : BOOL ;
    Alarm51 : BOOL ;
    Alarm52 : BOOL ;
    Alarm53 : BOOL ;
    Alarm54 : BOOL ;
    Alarm55 : BOOL ;
    Alarm56 : BOOL ;
    Alarm57 : BOOL ;
    Alarm58 : BOOL ;
    Alarm59 : BOOL ;
    Alarm60 : BOOL ;
    Alarm61 : BOOL ;
    Alarm62 : BOOL ;
    Alarm63 : BOOL ;
    Alarm64 : BOOL ;
   END_STRUCT ;
   StopCycle : STRUCT
    Alarm01 : BOOL ;	//Errore rilevamento anello di adattamento 1
    Alarm02 : BOOL ;	//Errore rilevamento anello di adattamento 2
    Alarm03 : BOOL ;	//Index cassetto non alto
    Alarm04 : BOOL ;	//Index cassetto non basso
    Alarm05 : BOOL ;	//Incongruenza sensori index cassetto
    Alarm06 : BOOL ;	//Cilindro sblocco pezzo non avanti
    Alarm07 : BOOL ;	//Cilindro sblocco pezzo non indietro
    Alarm08 : BOOL ;	//Incongruenza sensori cilindro sblocco pezzo
    Alarm09 : BOOL ;	//OP10 ToolType error
    Alarm10 : BOOL ;	//OP10 ToolCode error
    Alarm11 : BOOL ;
    Alarm12 : BOOL ;
    Alarm13 : BOOL ;
    Alarm14 : BOOL ;
    Alarm15 : BOOL ;
    Alarm16 : BOOL ;
    Alarm17 : BOOL ;
    Alarm18 : BOOL ;
    Alarm19 : BOOL ;
    Alarm20 : BOOL ;
    Alarm21 : BOOL ;
    Alarm22 : BOOL ;
    Alarm23 : BOOL ;
    Alarm24 : BOOL ;
    Alarm25 : BOOL ;
    Alarm26 : BOOL ;
    Alarm27 : BOOL ;
    Alarm28 : BOOL ;
    Alarm29 : BOOL ;
    Alarm30 : BOOL ;
    Alarm31 : BOOL ;
    Alarm32 : BOOL ;
    Alarm33 : BOOL ;
    Alarm34 : BOOL ;
    Alarm35 : BOOL ;
    Alarm36 : BOOL ;
    Alarm37 : BOOL ;
    Alarm38 : BOOL ;
    Alarm39 : BOOL ;
    Alarm40 : BOOL ;
    Alarm41 : BOOL ;
    Alarm42 : BOOL ;
    Alarm43 : BOOL ;
    Alarm44 : BOOL ;
    Alarm45 : BOOL ;
    Alarm46 : BOOL ;
    Alarm47 : BOOL ;
    Alarm48 : BOOL ;
    Alarm49 : BOOL ;
    Alarm50 : BOOL ;
    Alarm51 : BOOL ;
    Alarm52 : BOOL ;
    Alarm53 : BOOL ;
    Alarm54 : BOOL ;
    Alarm55 : BOOL ;
    Alarm56 : BOOL ;
    Alarm57 : BOOL ;
    Alarm58 : BOOL ;
    Alarm59 : BOOL ;
    Alarm60 : BOOL ;
    Alarm61 : BOOL ;
    Alarm62 : BOOL ;
    Alarm63 : BOOL ;
    Alarm64 : BOOL ;
   END_STRUCT ;
   RestartCycle : STRUCT
    Alarm01 : BOOL ;
    Alarm02 : BOOL ;
    Alarm03 : BOOL ;
    Alarm04 : BOOL ;
    Alarm05 : BOOL ;
    Alarm06 : BOOL ;
    Alarm07 : BOOL ;
    Alarm08 : BOOL ;
    Alarm09 : BOOL ;
    Alarm10 : BOOL ;
    Alarm11 : BOOL ;
    Alarm12 : BOOL ;
    Alarm13 : BOOL ;
    Alarm14 : BOOL ;
    Alarm15 : BOOL ;
    Alarm16 : BOOL ;
    Alarm17 : BOOL ;
    Alarm18 : BOOL ;
    Alarm19 : BOOL ;
    Alarm20 : BOOL ;
    Alarm21 : BOOL ;
    Alarm22 : BOOL ;
    Alarm23 : BOOL ;
    Alarm24 : BOOL ;
    Alarm25 : BOOL ;
    Alarm26 : BOOL ;
    Alarm27 : BOOL ;
    Alarm28 : BOOL ;
    Alarm29 : BOOL ;
    Alarm30 : BOOL ;
    Alarm31 : BOOL ;
    Alarm32 : BOOL ;
    Alarm33 : BOOL ;
    Alarm34 : BOOL ;
    Alarm35 : BOOL ;
    Alarm36 : BOOL ;
    Alarm37 : BOOL ;
    Alarm38 : BOOL ;
    Alarm39 : BOOL ;
    Alarm40 : BOOL ;
    Alarm41 : BOOL ;
    Alarm42 : BOOL ;
    Alarm43 : BOOL ;
    Alarm44 : BOOL ;
    Alarm45 : BOOL ;
    Alarm46 : BOOL ;
    Alarm47 : BOOL ;
    Alarm48 : BOOL ;
    Alarm49 : BOOL ;
    Alarm50 : BOOL ;
    Alarm51 : BOOL ;
    Alarm52 : BOOL ;
    Alarm53 : BOOL ;
    Alarm54 : BOOL ;
    Alarm55 : BOOL ;
    Alarm56 : BOOL ;
    Alarm57 : BOOL ;
    Alarm58 : BOOL ;
    Alarm59 : BOOL ;
    Alarm60 : BOOL ;
    Alarm61 : BOOL ;
    Alarm62 : BOOL ;
    Alarm63 : BOOL ;
    Alarm64 : BOOL ;
   END_STRUCT ;
   Warning : STRUCT
    Alarm01 : BOOL ;	//Blocco movimento index cassetto se cassetto non dentro o non fuori
    Alarm02 : BOOL ;	//Blocco sblocco pezzo se cassetto non fuori
    Alarm03 : BOOL ;	//Sblocco index solo con ribaditrice alta
    Alarm04 : BOOL ;	//Sblocco index solo con assi fermi
    Alarm05 : BOOL ;	//Sblocco index solo pezzo bloccato
    Alarm06 : BOOL ;
    Alarm07 : BOOL ;
    Alarm08 : BOOL ;
    Alarm09 : BOOL ;
    Alarm10 : BOOL ;
    Alarm11 : BOOL ;
    Alarm12 : BOOL ;
    Alarm13 : BOOL ;
    Alarm14 : BOOL ;
    Alarm15 : BOOL ;
    Alarm16 : BOOL ;
    Alarm17 : BOOL ;
    Alarm18 : BOOL ;
    Alarm19 : BOOL ;
    Alarm20 : BOOL ;
    Alarm21 : BOOL ;
    Alarm22 : BOOL ;
    Alarm23 : BOOL ;
    Alarm24 : BOOL ;
    Alarm25 : BOOL ;
    Alarm26 : BOOL ;
    Alarm27 : BOOL ;
    Alarm28 : BOOL ;
    Alarm29 : BOOL ;
    Alarm30 : BOOL ;
    Alarm31 : BOOL ;
    Alarm32 : BOOL ;
    Alarm33 : BOOL ;
    Alarm34 : BOOL ;
    Alarm35 : BOOL ;
    Alarm36 : BOOL ;
    Alarm37 : BOOL ;
    Alarm38 : BOOL ;
    Alarm39 : BOOL ;
    Alarm40 : BOOL ;
    Alarm41 : BOOL ;
    Alarm42 : BOOL ;
    Alarm43 : BOOL ;
    Alarm44 : BOOL ;
    Alarm45 : BOOL ;
    Alarm46 : BOOL ;
    Alarm47 : BOOL ;
    Alarm48 : BOOL ;
    Alarm49 : BOOL ;
    Alarm50 : BOOL ;
    Alarm51 : BOOL ;
    Alarm52 : BOOL ;
    Alarm53 : BOOL ;
    Alarm54 : BOOL ;
    Alarm55 : BOOL ;
    Alarm56 : BOOL ;
    Alarm57 : BOOL ;
    Alarm58 : BOOL ;
    Alarm59 : BOOL ;
    Alarm60 : BOOL ;
    Alarm61 : BOOL ;
    Alarm62 : BOOL ;
    Alarm63 : BOOL ;
    Alarm64 : BOOL ;
   END_STRUCT ;
  END_STRUCT ;	
BEGIN
END_DATA_BLOCK

DATA_BLOCK "Op10.Bench.Systems"	// DB 105
VERSION : 0.1
  STRUCT
   Command : STRUCT 	//
    Reset_allarmi : BOOL ;
    TestLampade : BOOL ;
    Abbassa_index_cassetto : BOOL ;
    Alza_index_cassetto : BOOL ;
    Sblocca_pezzo : BOOL ;
    Blocca_pezzo : BOOL ;
    FP_Consenso_operatore : BOOL ;
    Prenota_ribaditrice : BOOL ;
    Vai_in_posizione_assi : BOOL ;
    Marcia_ribaditrice : BOOL ;
    Abbassa_ribaditrice : BOOL ;
    Alza_ribaditrice : BOOL ;
    ris_w2 : DWORD ;
    ris_w6 : DWORD ;
   END_STRUCT ;
   State : STRUCT
    Porte_chiuse : BOOL ;
    Porte_chiuse_e_bloccate : BOOL ;
    Cassetto_dentro : BOOL ;
    Cassetto_fuori : BOOL ;
    Index_cassetto_basso : BOOL ;
    Index_cassetto_alto : BOOL ;
    Pezzo_sbloccato : BOOL ;
    Pezzo_bloccato : BOOL ;
    _Ribaditrice_a_disposiz : BOOL ;
    _Assi_posiz_raggiunta : BOOL ;
    Ribaditura_effettuata : BOOL ;
    Ribaditrice_alta : BOOL ;
    Ribaditrice_bassa : BOOL ;
    Ribaditrice_in_marcia : BOOL ;
    FP_stato_20_generale : BOOL ;
    _Ribad_in_fuori_ingombro : BOOL ;
    FP_Mode_automatic : BOOL ;
    FP_uscita_da_allarme : BOOL ;
    Ribaditura_pezzo_OK : BOOL ;
    Ribaditura_pezzo_KO : BOOL ;
    Assi_fermi : BOOL ;
    ris_w4 : WORD ;
    ris_w6 : DWORD ;
   END_STRUCT ;
   Data : STRUCT
    Num_punto_in_lavorazione : INT ;
    Pos_comandata_asse_X : DINT ;	//Punto in lavorazione
    Pos_comandata_asse_Y : DINT ;	//Punto in lavorazione
    Tempo_ribaditura : DINT ;	//Punto in lavorazione
    ris_w2 : DWORD ;
    ris_w6 : DWORD ;
   END_STRUCT ;
  END_STRUCT ;	
BEGIN
END_DATA_BLOCK

DATA_BLOCK "Op10.Tools.MapE"	// DB 106
VERSION : 0.1
  STRUCT
   ToolCode_Bit_0 : BOOL ;	//
   ToolCode_Bit_1 : BOOL ;
   ToolCode_Bit_2 : BOOL ;
   ToolCode_Bit_3 : BOOL ;
   ToolCode_Bit_4 : BOOL ;
   Anello_1_Inserito : BOOL ;
   Anello_2_Inserito : BOOL ;
   Presenza_nozzle_ring : BOOL ;
   Spacer_1_presente : BOOL ;
   Spacer_1_invertito : BOOL ;
   Spacer_2_presente : BOOL ;
   Spacer_2_invertito : BOOL ;
   Spacer_3_presente : BOOL ;
   Spacer_3_invertito : BOOL ;
   Ris_1_6 : BOOL ;
   Ris_1_7 : BOOL ;
  END_STRUCT ;	
BEGIN
END_DATA_BLOCK

DATA_BLOCK "Op10.Tools.Config"	// DB 108
VERSION : 0.1
  STRUCT
   DB_VAR : INT ;	//Variabile jolly provvisoria
  END_STRUCT ;	
BEGIN
END_DATA_BLOCK

DATA_BLOCK "Op10.Bench.Recipe"	// DB 110
VERSION : 0.1
  STRUCT
   ID_Ricetta : INT ;
   PartNumber : ARRAY  [0 .. 31 ] OF //Part number in lavorazione
   CHAR ;
   ToolType : INT ;	//Tool type
   ToolCode : INT ;	//Codice su attrezzo - ingressi digitali
   Anello1Abilitato : BOOL ;
   Anello2Abilitato : BOOL ;
   Velocita_asse_X : DINT ;
   Velocita_asse_Y : DINT ;
   spare48 : DINT ;
   spare52 : DINT ;
   spare56 : DINT ;
   spare60 : DINT ;
   spare64 : DINT ;
   spare68 : DINT ;
   spare72 : DINT ;
   spare76 : INT ;
   Disable : STRUCT 	//da indirizzo 78
    CkCodicePortapezzo : BOOL ;
    CkPresAnelloAdattamento : BOOL ;
    CkPresenzaNozzleRing : BOOL ;
    CkPresenzaSpacer1 : BOOL ;
    CkPresenzaSpacer2 : BOOL ;
    CkPresenzaSpacer3 : BOOL ;
    CheckSpare1 : BOOL ;
    CheckSpare2 : BOOL ;
    CheckSpare3 : BOOL ;
    CheckSpare4 : BOOL ;
   END_STRUCT ;
   NumeroPosizioni : INT ;
   posizioni : ARRAY  [0 .. 19 ] OF //da indirizzo 82
   STRUCT
    X : DINT ;	//1/100 mm
    Y : DINT ;	//1/100 mm
    TempoRibaditura : DINT ;	//msec
   END_STRUCT ;
   spare : ARRAY  [0 .. 38 ] OF INT ;
  END_STRUCT ;	
BEGIN
   PartNumber[0] := ' ';
   PartNumber[1] := ' ';
   PartNumber[2] := ' ';
   PartNumber[3] := ' ';
   PartNumber[4] := ' ';
   PartNumber[5] := ' ';
   PartNumber[6] := ' ';
   PartNumber[7] := ' ';
   PartNumber[8] := ' ';
   PartNumber[9] := ' ';
   PartNumber[10] := ' ';
   PartNumber[11] := ' ';
   PartNumber[12] := ' ';
   PartNumber[13] := ' ';
   PartNumber[14] := ' ';
   PartNumber[15] := ' ';
   PartNumber[16] := ' ';
   PartNumber[17] := ' ';
   PartNumber[18] := ' ';
   PartNumber[19] := ' ';
   PartNumber[20] := ' ';
   PartNumber[21] := ' ';
   PartNumber[22] := ' ';
   PartNumber[23] := ' ';
   PartNumber[24] := ' ';
   PartNumber[25] := ' ';
   PartNumber[26] := ' ';
   PartNumber[27] := ' ';
   PartNumber[28] := ' ';
   PartNumber[29] := ' ';
   PartNumber[30] := ' ';
   PartNumber[31] := ' ';
END_DATA_BLOCK

DATA_BLOCK "Op10.Cycles"	// DB 120
VERSION : 0.1
  STRUCT
   General : UDT 200;
   Restore : UDT 200;
  END_STRUCT ;	
BEGIN
END_DATA_BLOCK

DATA_BLOCK "OP20"	// DB 150
VERSION : 0.1
  STRUCT
   Mode : STRUCT
    Emergency : BOOL ;	//MODO Macchina spenta
    Test_Machine : BOOL ;	//MODO Aspetta pressione nel circuito pneumatico e/o idraulico + MODO Test Lampad
    Setup : BOOL ;	//MODO Cambio Ricetta o setup
    Manual : BOOL ;	//MODO Manuale
    Automatic : BOOL ;	//MODO Automatico
    Service : BOOL ;	//MODO Messa in servizio
    Free_06 : BOOL ;
    Free_07 : BOOL ;
   END_STRUCT ;
   Diagnostic : STRUCT
    Alarm_Emergency : BOOL ;	//Macchina in Emergenza
    Alarm_Stop_Cycle : BOOL ;	//Allarme che blocca il ciclo attivo
    Alarm_No_Restart : BOOL ;	//Allarme che blocca un nuovo ciclo
    Alarm_Warning : BOOL ;	//Segnalazione o avvertenza
    Safe_State : BOOL ;	//MODO Sicuro : e' possibile eseguire i comandi manuali in sicurezza
    Initial_Conditions : BOOL ;	//condizioni iniziali macchina
    Hold_State : BOOL ;	//Hold Macchina
    Free_07 : BOOL ;
    ResetAlarm : BOOL ;
   END_STRUCT ;
   Software : STRUCT
    SwName : STRING  [20 ];
    SwVersion : STRING  [11 ];
   END_STRUCT ;
  END_STRUCT ;	
BEGIN
END_DATA_BLOCK

DATA_BLOCK "Op20.Bench.MapE"	// DB 151
VERSION : 0.1
  STRUCT
   Ris_0_0 : BOOL ;
   Ris_0_1 : BOOL ;
   Cassetto_dentro : BOOL ;	//manca ingresso
   Index_cassetto_Giu : BOOL ;	//manca ingresso
   Index_cassetto_Su : BOOL ;	//manca ingresso
   Piantaggio_Giu : BOOL ;
   Piantaggio_Su : BOOL ;
   Gruppo_piantaggio_Giu : BOOL ;
   Gruppo_piantaggio_Su : BOOL ;
   Ris_w2 : WORD ;
   ris_w3 : WORD ;
   _Posizione_Punzone : REAL ;	//mm
  END_STRUCT ;	
BEGIN
END_DATA_BLOCK

DATA_BLOCK "Op20.Bench.MapA"	// DB 152
VERSION : 0.1
  STRUCT
   Fine_ciclo_OK : BOOL ;	//
   Fine_ciclo_NON_OK : BOOL ;
   EV_abb_index_cassetto : BOOL ;	//Libera index cassetto su zona piantaggio
   EV_alza_index_cassetto : BOOL ;	//Blocca index cassetto su zona piantaggio
   EV_abbassa_piantaggio : BOOL ;
   EV_alza_piantaggio : BOOL ;
   EV_abb_grupp_piantaggio : BOOL ;
   EV_alz_grupp_piantaggio : BOOL ;
  END_STRUCT ;	
BEGIN
END_DATA_BLOCK

DATA_BLOCK "Op20.Bench.Config"	// DB 153
VERSION : 0.1
  STRUCT
   Offset_Tastatore : REAL ;	//
  END_STRUCT ;	
BEGIN
END_DATA_BLOCK

DATA_BLOCK "Op20.Bench.Alarms"	// DB 154
VERSION : 0.1
  STRUCT
   Emegency : STRUCT
    Alarm01 : BOOL ;	//OP20 ToolType error
    Alarm02 : BOOL ;	//OP20 ToolCode error
    Alarm03 : BOOL ;
    Alarm04 : BOOL ;
    Alarm05 : BOOL ;
    Alarm06 : BOOL ;
    Alarm07 : BOOL ;
    Alarm08 : BOOL ;
    Alarm09 : BOOL ;	//
    Alarm10 : BOOL ;	//
    Alarm11 : BOOL ;	//
    Alarm12 : BOOL ;	//
    Alarm13 : BOOL ;	//
    Alarm14 : BOOL ;	//
    Alarm15 : BOOL ;
    Alarm16 : BOOL ;
    Alarm17 : BOOL ;
    Alarm18 : BOOL ;
    Alarm19 : BOOL ;
    Alarm20 : BOOL ;
    Alarm21 : BOOL ;
    Alarm22 : BOOL ;
    Alarm23 : BOOL ;
    Alarm24 : BOOL ;
    Alarm25 : BOOL ;
    Alarm26 : BOOL ;
    Alarm27 : BOOL ;
    Alarm28 : BOOL ;
    Alarm29 : BOOL ;
    Alarm30 : BOOL ;
    Alarm31 : BOOL ;
    Alarm32 : BOOL ;
    Alarm33 : BOOL ;
    Alarm34 : BOOL ;
    Alarm35 : BOOL ;
    Alarm36 : BOOL ;
    Alarm37 : BOOL ;
    Alarm38 : BOOL ;
    Alarm39 : BOOL ;
    Alarm40 : BOOL ;
    Alarm41 : BOOL ;
    Alarm42 : BOOL ;
    Alarm43 : BOOL ;
    Alarm44 : BOOL ;
    Alarm45 : BOOL ;
    Alarm46 : BOOL ;
    Alarm47 : BOOL ;
    Alarm48 : BOOL ;
    Alarm49 : BOOL ;
    Alarm50 : BOOL ;
    Alarm51 : BOOL ;
    Alarm52 : BOOL ;
    Alarm53 : BOOL ;
    Alarm54 : BOOL ;
    Alarm55 : BOOL ;
    Alarm56 : BOOL ;
    Alarm57 : BOOL ;
    Alarm58 : BOOL ;
    Alarm59 : BOOL ;
    Alarm60 : BOOL ;
    Alarm61 : BOOL ;
    Alarm62 : BOOL ;
    Alarm63 : BOOL ;
    Alarm64 : BOOL ;
   END_STRUCT ;
   StopCycle : STRUCT
    Alarm01 : BOOL ;	//Gruppo di piantaggio non basso
    Alarm02 : BOOL ;	//Gruppo di piantaggio non alto
    Alarm03 : BOOL ;	//Incongruenza sensori gruppo di piantaggio
    Alarm04 : BOOL ;	//piantaggio non basso
    Alarm05 : BOOL ;	//piantaggio non alto
    Alarm06 : BOOL ;	//Incongruenza sensori piantaggio
    Alarm07 : BOOL ;	//OP20 ToolType error
    Alarm08 : BOOL ;	//OP20 ToolCode error
    Alarm09 : BOOL ;
    Alarm10 : BOOL ;
    Alarm11 : BOOL ;
    Alarm12 : BOOL ;
    Alarm13 : BOOL ;
    Alarm14 : BOOL ;
    Alarm15 : BOOL ;
    Alarm16 : BOOL ;
    Alarm17 : BOOL ;
    Alarm18 : BOOL ;
    Alarm19 : BOOL ;
    Alarm20 : BOOL ;
    Alarm21 : BOOL ;
    Alarm22 : BOOL ;
    Alarm23 : BOOL ;
    Alarm24 : BOOL ;
    Alarm25 : BOOL ;
    Alarm26 : BOOL ;
    Alarm27 : BOOL ;
    Alarm28 : BOOL ;
    Alarm29 : BOOL ;
    Alarm30 : BOOL ;
    Alarm31 : BOOL ;
    Alarm32 : BOOL ;
    Alarm33 : BOOL ;
    Alarm34 : BOOL ;
    Alarm35 : BOOL ;
    Alarm36 : BOOL ;
    Alarm37 : BOOL ;
    Alarm38 : BOOL ;
    Alarm39 : BOOL ;
    Alarm40 : BOOL ;
    Alarm41 : BOOL ;
    Alarm42 : BOOL ;
    Alarm43 : BOOL ;
    Alarm44 : BOOL ;
    Alarm45 : BOOL ;
    Alarm46 : BOOL ;
    Alarm47 : BOOL ;
    Alarm48 : BOOL ;
    Alarm49 : BOOL ;
    Alarm50 : BOOL ;
    Alarm51 : BOOL ;
    Alarm52 : BOOL ;
    Alarm53 : BOOL ;
    Alarm54 : BOOL ;
    Alarm55 : BOOL ;
    Alarm56 : BOOL ;
    Alarm57 : BOOL ;
    Alarm58 : BOOL ;
    Alarm59 : BOOL ;
    Alarm60 : BOOL ;
    Alarm61 : BOOL ;
    Alarm62 : BOOL ;
    Alarm63 : BOOL ;
    Alarm64 : BOOL ;
   END_STRUCT ;
   RestartCycle : STRUCT
    Alarm01 : BOOL ;
    Alarm02 : BOOL ;
    Alarm03 : BOOL ;
    Alarm04 : BOOL ;
    Alarm05 : BOOL ;
    Alarm06 : BOOL ;
    Alarm07 : BOOL ;
    Alarm08 : BOOL ;
    Alarm09 : BOOL ;
    Alarm10 : BOOL ;
    Alarm11 : BOOL ;
    Alarm12 : BOOL ;
    Alarm13 : BOOL ;
    Alarm14 : BOOL ;
    Alarm15 : BOOL ;
    Alarm16 : BOOL ;
    Alarm17 : BOOL ;
    Alarm18 : BOOL ;
    Alarm19 : BOOL ;
    Alarm20 : BOOL ;
    Alarm21 : BOOL ;
    Alarm22 : BOOL ;
    Alarm23 : BOOL ;
    Alarm24 : BOOL ;
    Alarm25 : BOOL ;
    Alarm26 : BOOL ;
    Alarm27 : BOOL ;
    Alarm28 : BOOL ;
    Alarm29 : BOOL ;
    Alarm30 : BOOL ;
    Alarm31 : BOOL ;
    Alarm32 : BOOL ;
    Alarm33 : BOOL ;
    Alarm34 : BOOL ;
    Alarm35 : BOOL ;
    Alarm36 : BOOL ;
    Alarm37 : BOOL ;
    Alarm38 : BOOL ;
    Alarm39 : BOOL ;
    Alarm40 : BOOL ;
    Alarm41 : BOOL ;
    Alarm42 : BOOL ;
    Alarm43 : BOOL ;
    Alarm44 : BOOL ;
    Alarm45 : BOOL ;
    Alarm46 : BOOL ;
    Alarm47 : BOOL ;
    Alarm48 : BOOL ;
    Alarm49 : BOOL ;
    Alarm50 : BOOL ;
    Alarm51 : BOOL ;
    Alarm52 : BOOL ;
    Alarm53 : BOOL ;
    Alarm54 : BOOL ;
    Alarm55 : BOOL ;
    Alarm56 : BOOL ;
    Alarm57 : BOOL ;
    Alarm58 : BOOL ;
    Alarm59 : BOOL ;
    Alarm60 : BOOL ;
    Alarm61 : BOOL ;
    Alarm62 : BOOL ;
    Alarm63 : BOOL ;
    Alarm64 : BOOL ;
   END_STRUCT ;
   Warning : STRUCT
    Alarm01 : BOOL ;	//Blocco movimento index cassetto se cassetto non dentro
    Alarm02 : BOOL ;	//Index cassetto non alto
    Alarm03 : BOOL ;	//Index cassetto non basso
    Alarm04 : BOOL ;	//Incongruenza sensori index cassetto
    Alarm05 : BOOL ;	//Blocco movimento index cassetto con Pinataggio non alto
    Alarm06 : BOOL ;	//Blocco discesa Piantaggio con cassetto non dentro
    Alarm07 : BOOL ;	//Blocco discesa Piantaggio con cassetto non indexato
    Alarm08 : BOOL ;	//Blocco discesa Piantaggio con gruppo non basso
    Alarm09 : BOOL ;	//Blocco salita Gr Piantaggio se Piantaggio non alto
    Alarm10 : BOOL ;
    Alarm11 : BOOL ;
    Alarm12 : BOOL ;
    Alarm13 : BOOL ;
    Alarm14 : BOOL ;
    Alarm15 : BOOL ;
    Alarm16 : BOOL ;
    Alarm17 : BOOL ;
    Alarm18 : BOOL ;
    Alarm19 : BOOL ;
    Alarm20 : BOOL ;
    Alarm21 : BOOL ;
    Alarm22 : BOOL ;
    Alarm23 : BOOL ;
    Alarm24 : BOOL ;
    Alarm25 : BOOL ;
    Alarm26 : BOOL ;
    Alarm27 : BOOL ;
    Alarm28 : BOOL ;
    Alarm29 : BOOL ;
    Alarm30 : BOOL ;
    Alarm31 : BOOL ;
    Alarm32 : BOOL ;
    Alarm33 : BOOL ;
    Alarm34 : BOOL ;
    Alarm35 : BOOL ;
    Alarm36 : BOOL ;
    Alarm37 : BOOL ;
    Alarm38 : BOOL ;
    Alarm39 : BOOL ;
    Alarm40 : BOOL ;
    Alarm41 : BOOL ;
    Alarm42 : BOOL ;
    Alarm43 : BOOL ;
    Alarm44 : BOOL ;
    Alarm45 : BOOL ;
    Alarm46 : BOOL ;
    Alarm47 : BOOL ;
    Alarm48 : BOOL ;
    Alarm49 : BOOL ;
    Alarm50 : BOOL ;
    Alarm51 : BOOL ;
    Alarm52 : BOOL ;
    Alarm53 : BOOL ;
    Alarm54 : BOOL ;
    Alarm55 : BOOL ;
    Alarm56 : BOOL ;
    Alarm57 : BOOL ;
    Alarm58 : BOOL ;
    Alarm59 : BOOL ;
    Alarm60 : BOOL ;
    Alarm61 : BOOL ;
    Alarm62 : BOOL ;
    Alarm63 : BOOL ;
    Alarm64 : BOOL ;
   END_STRUCT ;
  END_STRUCT ;	
BEGIN
END_DATA_BLOCK

DATA_BLOCK "Op20.Bench.Systems"	// DB 155
VERSION : 0.1
  STRUCT
   Command : STRUCT 	//
    Reset_allarmi : BOOL ;
    TestLampade : BOOL ;
    Abbassa_index_cassetto : BOOL ;
    Alza_index_cassetto : BOOL ;
    Alza_gruppo_piantaggio : BOOL ;
    Abbasa_gruppo_piantaggio : BOOL ;
    Alza_piantaggio : BOOL ;
    Abbasa_piantaggio : BOOL ;
    ris_w2 : DWORD ;
    ris_w6 : DWORD ;
   END_STRUCT ;
   State : STRUCT 	//da indirizzo 10
    Porte_chiuse : BOOL ;
    Porte_chiuse_e_bloccate : BOOL ;
    Cassetto_dentro : BOOL ;
    Cassetto_fuori : BOOL ;
    Index_cassetto_basso : BOOL ;
    Index_cassetto_alto : BOOL ;
    Gruppo_piantaggio_alto : BOOL ;
    Gruppo_piantaggio_basso : BOOL ;
    Piantaggio_alto : BOOL ;
    Piantaggio_basso : BOOL ;
    Piantaggiofinito : BOOL ;
    Piantaggio_pezzo_OK : BOOL ;
    Piantaggio_pezzo_KO : BOOL ;
    FP_Mode_automatic : BOOL ;
    FP_uscita_da_allarme : BOOL ;
    FP_Cassettodentro : BOOL ;
    CassetDentroInizioCiclo : BOOL ;
    ris_w24 : WORD ;
    ris_w6 : DWORD ;
   END_STRUCT ;
   Data : STRUCT 	//da indirizzo 20
    frr1 : BOOL ;
    ris_w2 : DWORD ;
    ris_w6 : DWORD ;
   END_STRUCT ;
  END_STRUCT ;	
BEGIN
END_DATA_BLOCK

DATA_BLOCK "Op20.Tools.MapE"	// DB 156
VERSION : 0.1
  STRUCT
   ToolCode_Bit_0 : BOOL ;	//
   ToolCode_Bit_1 : BOOL ;
   ToolCode_Bit_2 : BOOL ;
   ToolCode_Bit_3 : BOOL ;
   ToolCode_Bit_4 : BOOL ;
   Ris_0_05 : BOOL ;
   Ris_0_06 : BOOL ;
   Ris_0_07 : BOOL ;
  END_STRUCT ;	
BEGIN
END_DATA_BLOCK

DATA_BLOCK "Op20.Tools.Config"	// DB 158
VERSION : 0.1
  STRUCT
   DB_VAR : INT ;	//Variabile jolly provvisoria
  END_STRUCT ;	
BEGIN
END_DATA_BLOCK

DATA_BLOCK "Op20.Bench.Recipe"	// DB 160
VERSION : 0.1
  STRUCT
   ID_Ricetta : INT ;
   PartNumber : ARRAY  [0 .. 31 ] OF //Part number in lavorazione
   CHAR ;
   ToolType : INT ;	//Tool type
   ToolCode : INT ;	//Codice su attrezzo - ingressi digitali
   spare38 : DINT ;
   spare42 : DINT ;
   spare46 : DINT ;
   spare50 : ARRAY  [0 .. 13 ] OF INT ;
   Disable : STRUCT 	//da indirizzo 78
    CkCodicePortapezzo : BOOL ;
    CheckSpare50_1 : BOOL ;
    CheckSpare50_2 : BOOL ;
    CheckSpare50_3 : BOOL ;
    CheckSpare50_4 : BOOL ;
    CheckSpare50_5 : BOOL ;
    CheckSpare50_6 : BOOL ;
    CheckSpare50_7 : BOOL ;
    CheckSpare51_0 : BOOL ;
    CheckSpare51_1 : BOOL ;
   END_STRUCT ;
   Corsa_piantaggio_min : REAL ;	//mm
   Corsa_piantaggio_max : REAL ;	//mm
   Spare_88 : REAL ;	//
   Tempo_stabilizzazione : DINT ;	//Millisecondi
   Timeout_piantaggio : DINT ;	//millisecondi
   spare100 : INT ;
   spare102 : INT ;
   spare104 : INT ;
   spare106 : INT ;
   spare108 : INT ;
   spare110 : ARRAY  [0 .. 145 ] OF INT ;
  END_STRUCT ;	
BEGIN
   PartNumber[0] := ' ';
   PartNumber[1] := ' ';
   PartNumber[2] := ' ';
   PartNumber[3] := ' ';
   PartNumber[4] := ' ';
   PartNumber[5] := ' ';
   PartNumber[6] := ' ';
   PartNumber[7] := ' ';
   PartNumber[8] := ' ';
   PartNumber[9] := ' ';
   PartNumber[10] := ' ';
   PartNumber[11] := ' ';
   PartNumber[12] := ' ';
   PartNumber[13] := ' ';
   PartNumber[14] := ' ';
   PartNumber[15] := ' ';
   PartNumber[16] := ' ';
   PartNumber[17] := ' ';
   PartNumber[18] := ' ';
   PartNumber[19] := ' ';
   PartNumber[20] := ' ';
   PartNumber[21] := ' ';
   PartNumber[22] := ' ';
   PartNumber[23] := ' ';
   PartNumber[24] := ' ';
   PartNumber[25] := ' ';
   PartNumber[26] := ' ';
   PartNumber[27] := ' ';
   PartNumber[28] := ' ';
   PartNumber[29] := ' ';
   PartNumber[30] := ' ';
   PartNumber[31] := ' ';
END_DATA_BLOCK

DATA_BLOCK "Op20.Cycles"	// DB 170
VERSION : 0.1
  STRUCT
   General : UDT 200;
   Restore : UDT 200;
  END_STRUCT ;	
BEGIN
END_DATA_BLOCK

DATA_BLOCK "OP40"	// DB 200
VERSION : 0.1
  STRUCT
   Mode : STRUCT
    Emergency : BOOL ;	//MODO Macchina spenta
    Test_Machine : BOOL ;	//MODO Aspetta pressione nel circuito pneumatico e/o idraulico + MODO Test Lampad
    Setup : BOOL ;	//MODO Cambio Ricetta o setup
    Manual : BOOL ;	//MODO Manuale
    Automatic : BOOL ;	//MODO Automatico
    Service : BOOL ;	//MODO Messa in servizio
    Free_06 : BOOL ;
    Free_07 : BOOL ;
   END_STRUCT ;
   Diagnostic : STRUCT
    Alarm_Emergency : BOOL ;	//Macchina in Emergenza
    Alarm_Stop_Cycle : BOOL ;	//Allarme che blocca il ciclo attivo
    Alarm_No_Restart : BOOL ;	//Allarme che blocca un nuovo ciclo
    Alarm_Warning : BOOL ;	//Segnalazione o avvertenza
    Safe_State : BOOL ;	//MODO Sicuro : e' possibile eseguire i comandi manuali in sicurezza
    Initial_Conditions : BOOL ;	//condizioni iniziali macchina
    Hold_State : BOOL ;	//Hold Macchina
    Free_07 : BOOL ;
    ResetAlarm : BOOL ;
   END_STRUCT ;
   Software : STRUCT
    SwName : STRING  [20 ];
    SwVersion : STRING  [11 ];
   END_STRUCT ;
  END_STRUCT ;	
BEGIN
END_DATA_BLOCK

DATA_BLOCK "Op40.Bench.MapE"	// DB 201
VERSION : 0.1
  STRUCT
   PLS_Operator_confirm : BOOL ;	//(start ciclo)
   Pipe_placed : BOOL ;
   Box_out : BOOL ;
   Box_in : BOOL ;
   Box_index_up : BOOL ;
   Box_index_down : BOOL ;
   Unlock_parts_down : BOOL ;
   Unlock_parts_up : BOOL ;
   PLS_Stop_Cycle : BOOL ;
   Ring_lock_pipe_present : BOOL ;
   free001 : BOOL ;
   free002 : BOOL ;
   free003 : BOOL ;
   free004 : BOOL ;
   free005 : BOOL ;
   free006 : BOOL ;
  END_STRUCT ;	
BEGIN
END_DATA_BLOCK

DATA_BLOCK "Op40.Bench.MapA"	// DB 202
VERSION : 0.1
  STRUCT
   Fine_ciclo_OK : BOOL ;	//
   Fine_ciclo_NON_OK : BOOL ;
   EV_abb_index_cassetto : BOOL ;	//Libera index cassetto su zona piantaggio
   EV_alza_index_cassetto : BOOL ;	//Blocca index cassetto su zona piantaggio
   EV_sblocco_pezzo : BOOL ;
   EV_blocco_pezzo : BOOL ;
  END_STRUCT ;	
BEGIN
END_DATA_BLOCK

DATA_BLOCK "Op40.Bench.Config"	// DB 203
VERSION : 0.1
  STRUCT
   Dummy : INT ;	//
  END_STRUCT ;	
BEGIN
END_DATA_BLOCK

DATA_BLOCK "Op40.Bench.Alarms"	// DB 204
VERSION : 0.1
  STRUCT
   Emegency : STRUCT
    Alarm01 : BOOL ;	//OP40 ToolType error
    Alarm02 : BOOL ;	//OP40 Tool Code error
    Alarm03 : BOOL ;
    Alarm04 : BOOL ;
    Alarm05 : BOOL ;
    Alarm06 : BOOL ;
    Alarm07 : BOOL ;
    Alarm08 : BOOL ;
    Alarm09 : BOOL ;	//
    Alarm10 : BOOL ;	//
    Alarm11 : BOOL ;	//
    Alarm12 : BOOL ;	//
    Alarm13 : BOOL ;	//
    Alarm14 : BOOL ;	//
    Alarm15 : BOOL ;
    Alarm16 : BOOL ;
    Alarm17 : BOOL ;
    Alarm18 : BOOL ;
    Alarm19 : BOOL ;
    Alarm20 : BOOL ;
    Alarm21 : BOOL ;
    Alarm22 : BOOL ;
    Alarm23 : BOOL ;
    Alarm24 : BOOL ;
    Alarm25 : BOOL ;
    Alarm26 : BOOL ;
    Alarm27 : BOOL ;
    Alarm28 : BOOL ;
    Alarm29 : BOOL ;
    Alarm30 : BOOL ;
    Alarm31 : BOOL ;
    Alarm32 : BOOL ;
    Alarm33 : BOOL ;
    Alarm34 : BOOL ;
    Alarm35 : BOOL ;
    Alarm36 : BOOL ;
    Alarm37 : BOOL ;
    Alarm38 : BOOL ;
    Alarm39 : BOOL ;
    Alarm40 : BOOL ;
    Alarm41 : BOOL ;
    Alarm42 : BOOL ;
    Alarm43 : BOOL ;
    Alarm44 : BOOL ;
    Alarm45 : BOOL ;
    Alarm46 : BOOL ;
    Alarm47 : BOOL ;
    Alarm48 : BOOL ;
    Alarm49 : BOOL ;
    Alarm50 : BOOL ;
    Alarm51 : BOOL ;
    Alarm52 : BOOL ;
    Alarm53 : BOOL ;
    Alarm54 : BOOL ;
    Alarm55 : BOOL ;
    Alarm56 : BOOL ;
    Alarm57 : BOOL ;
    Alarm58 : BOOL ;
    Alarm59 : BOOL ;
    Alarm60 : BOOL ;
    Alarm61 : BOOL ;
    Alarm62 : BOOL ;
    Alarm63 : BOOL ;
    Alarm64 : BOOL ;
   END_STRUCT ;
   StopCycle : STRUCT
    Alarm01 : BOOL ;	//Errore rilevamento anello di adattamento 1
    Alarm02 : BOOL ;	//Errore rilevamento anello di adattamento 2
    Alarm03 : BOOL ;	//Index cassetto non alto
    Alarm04 : BOOL ;	//Index cassetto non basso
    Alarm05 : BOOL ;	//Incongruenza sensori index cassetto
    Alarm06 : BOOL ;	//Cilindro sblocco pezzo non avanti
    Alarm07 : BOOL ;	//Cilindro sblocco pezzo non indietro
    Alarm08 : BOOL ;	//Incongruenza sensori cilindro sblocco pezzo
    Alarm09 : BOOL ;	//OP40 ToolType error
    Alarm10 : BOOL ;	//OP40 Tool Code error
    Alarm11 : BOOL ;
    Alarm12 : BOOL ;
    Alarm13 : BOOL ;
    Alarm14 : BOOL ;
    Alarm15 : BOOL ;
    Alarm16 : BOOL ;
    Alarm17 : BOOL ;
    Alarm18 : BOOL ;
    Alarm19 : BOOL ;
    Alarm20 : BOOL ;
    Alarm21 : BOOL ;
    Alarm22 : BOOL ;
    Alarm23 : BOOL ;
    Alarm24 : BOOL ;
    Alarm25 : BOOL ;
    Alarm26 : BOOL ;
    Alarm27 : BOOL ;
    Alarm28 : BOOL ;
    Alarm29 : BOOL ;
    Alarm30 : BOOL ;
    Alarm31 : BOOL ;
    Alarm32 : BOOL ;
    Alarm33 : BOOL ;
    Alarm34 : BOOL ;
    Alarm35 : BOOL ;
    Alarm36 : BOOL ;
    Alarm37 : BOOL ;
    Alarm38 : BOOL ;
    Alarm39 : BOOL ;
    Alarm40 : BOOL ;
    Alarm41 : BOOL ;
    Alarm42 : BOOL ;
    Alarm43 : BOOL ;
    Alarm44 : BOOL ;
    Alarm45 : BOOL ;
    Alarm46 : BOOL ;
    Alarm47 : BOOL ;
    Alarm48 : BOOL ;
    Alarm49 : BOOL ;
    Alarm50 : BOOL ;
    Alarm51 : BOOL ;
    Alarm52 : BOOL ;
    Alarm53 : BOOL ;
    Alarm54 : BOOL ;
    Alarm55 : BOOL ;
    Alarm56 : BOOL ;
    Alarm57 : BOOL ;
    Alarm58 : BOOL ;
    Alarm59 : BOOL ;
    Alarm60 : BOOL ;
    Alarm61 : BOOL ;
    Alarm62 : BOOL ;
    Alarm63 : BOOL ;
    Alarm64 : BOOL ;
   END_STRUCT ;
   RestartCycle : STRUCT
    Alarm01 : BOOL ;
    Alarm02 : BOOL ;
    Alarm03 : BOOL ;
    Alarm04 : BOOL ;
    Alarm05 : BOOL ;
    Alarm06 : BOOL ;
    Alarm07 : BOOL ;
    Alarm08 : BOOL ;
    Alarm09 : BOOL ;
    Alarm10 : BOOL ;
    Alarm11 : BOOL ;
    Alarm12 : BOOL ;
    Alarm13 : BOOL ;
    Alarm14 : BOOL ;
    Alarm15 : BOOL ;
    Alarm16 : BOOL ;
    Alarm17 : BOOL ;
    Alarm18 : BOOL ;
    Alarm19 : BOOL ;
    Alarm20 : BOOL ;
    Alarm21 : BOOL ;
    Alarm22 : BOOL ;
    Alarm23 : BOOL ;
    Alarm24 : BOOL ;
    Alarm25 : BOOL ;
    Alarm26 : BOOL ;
    Alarm27 : BOOL ;
    Alarm28 : BOOL ;
    Alarm29 : BOOL ;
    Alarm30 : BOOL ;
    Alarm31 : BOOL ;
    Alarm32 : BOOL ;
    Alarm33 : BOOL ;
    Alarm34 : BOOL ;
    Alarm35 : BOOL ;
    Alarm36 : BOOL ;
    Alarm37 : BOOL ;
    Alarm38 : BOOL ;
    Alarm39 : BOOL ;
    Alarm40 : BOOL ;
    Alarm41 : BOOL ;
    Alarm42 : BOOL ;
    Alarm43 : BOOL ;
    Alarm44 : BOOL ;
    Alarm45 : BOOL ;
    Alarm46 : BOOL ;
    Alarm47 : BOOL ;
    Alarm48 : BOOL ;
    Alarm49 : BOOL ;
    Alarm50 : BOOL ;
    Alarm51 : BOOL ;
    Alarm52 : BOOL ;
    Alarm53 : BOOL ;
    Alarm54 : BOOL ;
    Alarm55 : BOOL ;
    Alarm56 : BOOL ;
    Alarm57 : BOOL ;
    Alarm58 : BOOL ;
    Alarm59 : BOOL ;
    Alarm60 : BOOL ;
    Alarm61 : BOOL ;
    Alarm62 : BOOL ;
    Alarm63 : BOOL ;
    Alarm64 : BOOL ;
   END_STRUCT ;
   Warning : STRUCT
    Alarm01 : BOOL ;	//Blocco movimento index cassetto se cassetto non dentro o non fuori
    Alarm02 : BOOL ;	//Blocco sblocco pezzo se cassetto non fuori
    Alarm03 : BOOL ;	//Sblocco index solo con ribaditrice alta
    Alarm04 : BOOL ;	//Sblocco index solo con assi fermi
    Alarm05 : BOOL ;	//Sblocco index solo pezzo bloccato
    Alarm06 : BOOL ;
    Alarm07 : BOOL ;
    Alarm08 : BOOL ;
    Alarm09 : BOOL ;
    Alarm10 : BOOL ;
    Alarm11 : BOOL ;
    Alarm12 : BOOL ;
    Alarm13 : BOOL ;
    Alarm14 : BOOL ;
    Alarm15 : BOOL ;
    Alarm16 : BOOL ;
    Alarm17 : BOOL ;
    Alarm18 : BOOL ;
    Alarm19 : BOOL ;
    Alarm20 : BOOL ;
    Alarm21 : BOOL ;
    Alarm22 : BOOL ;
    Alarm23 : BOOL ;
    Alarm24 : BOOL ;
    Alarm25 : BOOL ;
    Alarm26 : BOOL ;
    Alarm27 : BOOL ;
    Alarm28 : BOOL ;
    Alarm29 : BOOL ;
    Alarm30 : BOOL ;
    Alarm31 : BOOL ;
    Alarm32 : BOOL ;
    Alarm33 : BOOL ;
    Alarm34 : BOOL ;
    Alarm35 : BOOL ;
    Alarm36 : BOOL ;
    Alarm37 : BOOL ;
    Alarm38 : BOOL ;
    Alarm39 : BOOL ;
    Alarm40 : BOOL ;
    Alarm41 : BOOL ;
    Alarm42 : BOOL ;
    Alarm43 : BOOL ;
    Alarm44 : BOOL ;
    Alarm45 : BOOL ;
    Alarm46 : BOOL ;
    Alarm47 : BOOL ;
    Alarm48 : BOOL ;
    Alarm49 : BOOL ;
    Alarm50 : BOOL ;
    Alarm51 : BOOL ;
    Alarm52 : BOOL ;
    Alarm53 : BOOL ;
    Alarm54 : BOOL ;
    Alarm55 : BOOL ;
    Alarm56 : BOOL ;
    Alarm57 : BOOL ;
    Alarm58 : BOOL ;
    Alarm59 : BOOL ;
    Alarm60 : BOOL ;
    Alarm61 : BOOL ;
    Alarm62 : BOOL ;
    Alarm63 : BOOL ;
    Alarm64 : BOOL ;
   END_STRUCT ;
  END_STRUCT ;	
BEGIN
END_DATA_BLOCK

DATA_BLOCK "Op40.Bench.Systems"	// DB 205
VERSION : 0.1
  STRUCT
   Command : STRUCT 	//
    Reset_allarmi : BOOL ;
    TestLampade : BOOL ;
    Abbassa_index_cassetto : BOOL ;
    Alza_index_cassetto : BOOL ;
    Sblocca_pezzo : BOOL ;
    Blocca_pezzo : BOOL ;
    FP_Consenso_operatore : BOOL ;
    Prenota_ribaditrice : BOOL ;
    Vai_in_posizione_assi : BOOL ;
    Marcia_ribaditrice : BOOL ;
    Abbassa_ribaditrice : BOOL ;
    Alza_ribaditrice : BOOL ;
    ris_w2 : DWORD ;
    ris_w6 : DWORD ;
   END_STRUCT ;
   State : STRUCT 	//da indirizzo 10
    Porte_chiuse : BOOL ;
    Porte_chiuse_e_bloccate : BOOL ;
    Cassetto_dentro : BOOL ;
    Cassetto_fuori : BOOL ;
    Index_cassetto_basso : BOOL ;
    Index_cassetto_alto : BOOL ;
    Pezzo_sbloccato : BOOL ;
    Pezzo_bloccato : BOOL ;
    _Ribaditrice_a_disposiz : BOOL ;
    _Assi_posiz_raggiunta : BOOL ;
    Ribaditura_effettuata : BOOL ;
    Ribaditrice_alta : BOOL ;
    Ribaditrice_bassa : BOOL ;
    Ribaditrice_in_marcia : BOOL ;
    FP_stato_20_generale : BOOL ;
    _Ribad_in_fuori_ingombro : BOOL ;
    FP_Mode_automatic : BOOL ;
    FP_uscita_da_allarme : BOOL ;
    Ribaditura_pezzo_OK : BOOL ;
    Ribaditura_pezzo_KO : BOOL ;
    Assi_fermi : BOOL ;
    ris_w4 : WORD ;
    ris_w6 : DWORD ;
   END_STRUCT ;
   Data : STRUCT 	//da indirizzo 20
    Num_punto_in_lavorazione : INT ;
    Pos_comandata_asse_X : DINT ;	//Punto in lavorazione
    Pos_comandata_asse_Y : DINT ;	//Punto in lavorazione
    Tempo_ribaditura : DINT ;	//Punto in lavorazione
    ris_w2 : DWORD ;
    ris_w6 : DWORD ;
   END_STRUCT ;
  END_STRUCT ;	
BEGIN
END_DATA_BLOCK

DATA_BLOCK "Op40.Tools.MapE"	// DB 206
VERSION : 0.1
  STRUCT
   ToolCode_Bit_0 : BOOL ;	//
   ToolCode_Bit_1 : BOOL ;
   ToolCode_Bit_2 : BOOL ;
   ToolCode_Bit_3 : BOOL ;
   ToolCode_Bit_4 : BOOL ;
   Anello_1_Inserito : BOOL ;
   Anello_2_Inserito : BOOL ;
   Presenza_pin_roller : BOOL ;
  END_STRUCT ;	
BEGIN
END_DATA_BLOCK

DATA_BLOCK "Op40.Tools.Config"	// DB 208
VERSION : 0.1
  STRUCT
   DB_VAR : INT ;	//Variabile jolly provvisoria
  END_STRUCT ;	
BEGIN
END_DATA_BLOCK

DATA_BLOCK "Op40.Tools.Systems"	// DB 209
VERSION : 0.1
  STRUCT
   DB_VAR : INT ;	//Variabile jolly provvisoria
  END_STRUCT ;	
BEGIN
END_DATA_BLOCK

DATA_BLOCK "Op40.Bench.Recipe"	// DB 210
VERSION : 0.1
  STRUCT
   ID_Ricetta : INT ;
   PartNumber : ARRAY  [0 .. 31 ] OF //Part number in lavorazione
   CHAR ;
   ToolType : INT ;	//Tool type
   ToolCode : INT ;	//Codice su attrezzo - ingressi digitali
   Anello1Abilitato : BOOL ;
   Anello2Abilitato : BOOL ;
   Velocita_asse_X1 : DINT ;
   Velocita_asse_Y1 : DINT ;
   spare48 : DINT ;
   spare52 : DINT ;
   spare56 : DINT ;
   spare60 : DINT ;
   spare64 : DINT ;
   spare68 : DINT ;
   spare72 : DINT ;
   spare76 : INT ;
   Disable : STRUCT 	//da indirizzo 78
    CkCodicePortapezzo : BOOL ;
    CkPresAnelloAdattamento : BOOL ;
    CkPresenzaNozzleRing : BOOL ;
    CkPresenzaPipe : BOOL ;
    CheckSpare4 : BOOL ;
    CheckSpare5 : BOOL ;
    CheckSpare6 : BOOL ;
    CheckSpare7 : BOOL ;
    CheckSpare8 : BOOL ;
    CheckSpare9 : BOOL ;
   END_STRUCT ;
   NumeroPosizioni : INT ;
   posizioni : ARRAY  [0 .. 19 ] OF //da indirizzo 82
   STRUCT
    X : DINT ;	//1/100 mm
    Y : DINT ;	//1/100 mm
    TempoRibaditura : DINT ;	//msec
   END_STRUCT ;
   spare : ARRAY  [0 .. 38 ] OF INT ;
  END_STRUCT ;	
BEGIN
   PartNumber[0] := ' ';
   PartNumber[1] := ' ';
   PartNumber[2] := ' ';
   PartNumber[3] := ' ';
   PartNumber[4] := ' ';
   PartNumber[5] := ' ';
   PartNumber[6] := ' ';
   PartNumber[7] := ' ';
   PartNumber[8] := ' ';
   PartNumber[9] := ' ';
   PartNumber[10] := ' ';
   PartNumber[11] := ' ';
   PartNumber[12] := ' ';
   PartNumber[13] := ' ';
   PartNumber[14] := ' ';
   PartNumber[15] := ' ';
   PartNumber[16] := ' ';
   PartNumber[17] := ' ';
   PartNumber[18] := ' ';
   PartNumber[19] := ' ';
   PartNumber[20] := ' ';
   PartNumber[21] := ' ';
   PartNumber[22] := ' ';
   PartNumber[23] := ' ';
   PartNumber[24] := ' ';
   PartNumber[25] := ' ';
   PartNumber[26] := ' ';
   PartNumber[27] := ' ';
   PartNumber[28] := ' ';
   PartNumber[29] := ' ';
   PartNumber[30] := ' ';
   PartNumber[31] := ' ';
END_DATA_BLOCK

DATA_BLOCK "Op40.Cycles"	// DB 220
VERSION : 0.1
  STRUCT
   General : UDT 200;
   Restore : UDT 200;
  END_STRUCT ;	
BEGIN
END_DATA_BLOCK

DATA_BLOCK DB 400
VERSION : 0.0
"Std System.Cylinder"
BEGIN
END_DATA_BLOCK

DATA_BLOCK "Ist_cil_10_Index_cass"	// DB 401
VERSION : 0.0
"Std System.Cylinder"
BEGIN
END_DATA_BLOCK

DATA_BLOCK "Ist_10_CilBloccoPezzo"	// DB 402
VERSION : 0.0
"Std System.Cylinder"
BEGIN
END_DATA_BLOCK

DATA_BLOCK "Ist_cil_20_Index_cass"	// DB 403
VERSION : 0.0
"Std System.Cylinder"
BEGIN
END_DATA_BLOCK

DATA_BLOCK "Ist_cil_20_gr_piantaggio"	// DB 404
VERSION : 0.0
"Std System.Cylinder"
BEGIN
END_DATA_BLOCK

DATA_BLOCK "Ist_cil_20_piantaggio"	// DB 405
VERSION : 0.0
"Std System.Cylinder"
BEGIN
END_DATA_BLOCK

DATA_BLOCK "Ist_cil_40_Index_cass"	// DB 406
VERSION : 0.0
"Std System.Cylinder"
BEGIN
END_DATA_BLOCK

DATA_BLOCK "Ist_40_CilBloccoPezzo"	// DB 407
VERSION : 0.0
"Std System.Cylinder"
BEGIN
END_DATA_BLOCK

DATA_BLOCK "Ist_AsseX"	// DB 420
AUTHOR : Castel
VERSION : 0.0
"Std_Sinamics_Axis"
BEGIN
END_DATA_BLOCK

DATA_BLOCK "Ist_AsseY"	// DB 421
AUTHOR : Castel
VERSION : 0.0
"Std_Sinamics_Axis"
BEGIN
END_DATA_BLOCK

DATA_BLOCK "Ist_CU_asseX"	// DB 425
VERSION : 0.0
"Std.Sinamics_Cu_S"
BEGIN
END_DATA_BLOCK

DATA_BLOCK "Ist_CU_asseY"	// DB 426
VERSION : 0.0
"Std.Sinamics_Cu_S"
BEGIN
END_DATA_BLOCK

DATA_BLOCK "Op10.Ist.Cycle.General"	// DB 430
VERSION : 0.0
"Op10.Cycle.General"
BEGIN
END_DATA_BLOCK

DATA_BLOCK "Op10.Ist.Cycle.Restore"	// DB 431
VERSION : 0.0
"Op10.Cycle.Restore"
BEGIN
END_DATA_BLOCK

DATA_BLOCK "OP40.Ist.Cycle.Restore"	// DB 435
VERSION : 0.0
"Op40.Cycle.Restore"
BEGIN
END_DATA_BLOCK

DATA_BLOCK "OP40.Ist.Cycle.General"	// DB 436
VERSION : 0.0
"Op40.Cycle.General"
BEGIN
END_DATA_BLOCK

DATA_BLOCK "OP20.Ist.Cycle.Restore"	// DB 437
VERSION : 0.0
"Op20.Cycle.Restore"
BEGIN
END_DATA_BLOCK

DATA_BLOCK "OP20.Ist.Cycle.General"	// DB 438
VERSION : 0.0
"Op20.Cycle.General"
BEGIN
END_DATA_BLOCK

DATA_BLOCK "Line.Ist.Cycle.Coord_rib"	// DB 440
VERSION : 0.0
"Line.Cycle.Coord_ribadit"
BEGIN
END_DATA_BLOCK

ORGANIZATION_BLOCK OB 1
TITLE = "Main Program Sweep (Cycle)"
VERSION : 0.1
VAR_TEMP
  OB1_EV_CLASS : BYTE ;	//Bits 0-3 = 1 (Coming event), Bits 4-7 = 1 (Event class 1)
  OB1_SCAN_1 : BYTE ;	//1 (Cold restart scan 1 of OB 1), 3 (Scan 2-n of OB 1)
  OB1_PRIORITY : BYTE ;	//Priority of OB Execution
  OB1_OB_NUMBR : BYTE ;	//1 (Organization block 1, OB1)
  OB1_RESERVED_1 : BYTE ;	//Reserved for system
  OB1_RESERVED_2 : BYTE ;	//Reserved for system
  OB1_PREV_CYCLE : INT ;	//Cycle time of previous OB1 scan (milliseconds)
  OB1_MIN_CYCLE : INT ;	//Minimum cycle time of OB1 (milliseconds)
  OB1_MAX_CYCLE : INT ;	//Maximum cycle time of OB1 (milliseconds)
  OB1_DATE_TIME : DATE_AND_TIME ;	//Date and time OB1 started
END_VAR
BEGIN
NETWORK
TITLE = Bit Alw_ON e ALW_OFF
      SET;
      =     "Alw_ON";
      NOT;
      =     "alw_OFF";
NETWORK
TITLE = Line
      CALL  "Line.FCMain";
NETWORK
TITLE = OP10
      CALL  "OP10.FCMain";
NETWORK
TITLE = OP20
      CALL  "OP20.FCMain";
NETWORK
TITLE = op40
      CALL  "OP40.FCMain";
NETWORK
TITLE =
NETWORK
TITLE = Reset first scan
      CLR;
      =     "FirstScan";
END_ORGANIZATION_BLOCK

FUNCTION_BLOCK FB 60
VERSION : 0.1
VAR_INPUT
  IN_Cm_ON : BOOL ;	//1: Attiva il ciclo; 0: Reset del ciclo
  IN_HOLD : BOOL ;	//Blocca il ciclo nel passo successivo
  IN_STEP : BOOL ;
END_VAR
VAR_OUTPUT
  OUT_St_CicloInCorso : BOOL ;
  OUT_St_CicloTerminatoOK : BOOL ;
  OUT_St_CicloTerminatoKO : BOOL ;
  OUT_CicloStato : INT ;
  OUT_Page : INT ;
  OUT_Message : INT ;
END_VAR
VAR
  Stato : INT ;
  StatoSeguente : INT ;
  FrontePassoSingolo : BOOL ;
  Stat_CicloTermOk : BOOL ;
  Stat_CicloTermKO : BOOL ;
  Stat_CicloInCorso : BOOL ;
  Timer_Pennarello : SFB 4;
END_VAR
VAR_TEMP
  Pag_Active : ARRAY  [0 .. 100 ] OF BOOL ;
END_VAR
BEGIN
NETWORK
TITLE = FLOW CHART
NETWORK
TITLE = Update state
      A     #IN_Cm_ON;
      JC    M002;
      L     0;
      T     #Stato;
      T     #StatoSeguente;
M002: NOP   0;
//->Update State
      A     #IN_STEP;
      FP    #FrontePassoSingolo;
      ON    #IN_HOLD;	//se usassi UN l'Hold agirebbe anche su avanzamento a passo singolo 
      JCN   N100;
      L     #StatoSeguente;
      T     #Stato;
N100: NOP   0;
// determinazione bit di stato
      CALL  FC 17 (
           Valore                   := #Stato,
           States                   := P#DB60.DBX 8.0 BYTE 8);
NETWORK
TITLE = Detect page active from OP
// serve??????
//      CALL  "Conv_INT->BIT"
//       Valore:=DB325.DBW2
//       States:=#Pag_Active
NETWORK
TITLE = States particular
      L     #Stato;
      L     0;
      <>I;
//->Evita ritardi
      A     #IN_Cm_ON;
      =     #Stat_CicloInCorso;
      A     DB60.DBX 15.4;
      =     #Stat_CicloTermOk;
      A     DB60.DBX 15.7;
      =     #Stat_CicloTermKO;
NETWORK
TITLE = Diagnostic default
//    L     0
//    T     #Page
//    L     0
//    T     #Message 
//      L     6
//      T     #StatoSeguente
NETWORK
TITLE = State <0>: Ciclo off
      A     DB60.DBX 8.0;
      JCN   Z000;
      A     #IN_Cm_ON;
      A     DB55.DBX 3.0;
      JC    Y000;
      A     #IN_Cm_ON;
      A     DB55.DBX 3.1;
      JC    X000;
      JU    Z000;
Y000: L     10;
      T     #StatoSeguente;
      JU    Z000;
X000: L     20;
      T     #StatoSeguente;
Z000: NOP   0;
NETWORK
TITLE = State <10>: Ribaditrice prenotata da OP10
      A     DB60.DBX 9.2;
      JCN   Z010;
      AN    DB55.DBX 3.0;
      JC    Y010;
      JU    Z010;
// Stati di destinazione
Y010: L     0;
      T     #StatoSeguente;
Z010: NOP   0;
NETWORK
TITLE = State <20>: Ribaditrice prenotata da OP40
      A     DB60.DBX 10.4;
      JCN   Z020;
      AN    DB55.DBX 3.1;
      JC    Y020;
      JU    Z020;
// Stati di destinazione
Y020: L     0;
      T     #StatoSeguente;
Z020: NOP   0;
NETWORK
TITLE = Output
      L     #Stato;
      T     #OUT_CicloStato;
      A     #Stat_CicloInCorso;
      =     #OUT_St_CicloInCorso;
      A     #Stat_CicloTermOk;
      =     #OUT_St_CicloTerminatoOK;
      A     #Stat_CicloTermKO;
      =     #OUT_St_CicloTerminatoKO;
END_FUNCTION_BLOCK

FUNCTION_BLOCK FB 102
VERSION : 2.1
VAR_INPUT
  IN_Enable : BOOL ;	//Abilita/Disabilita le uscite e gli allarmi
  IN_Command_CylForward : BOOL ;	//Se a 1 e non in hold comanda l'elettrovalvola
  IN_Command_CylBack : BOOL ;	//Se a 1 e non in hold comanda l'elettrovalvola
  IN_EndStroke_Forward : BOOL ;	//Ingresso PLC E...
  IN_EndStroke_Back : BOOL ;	//Ingresso PLC E...
  IN_Alarms_Reset : BOOL ;	//Tasto di reset allarme (fronte interno)
  IN_Alarms_TimeOut : TIME ;	//Tempo in secondi per time-out rilevamento Fc dopo comando
  IN_Hold_Condition : BOOL ;	//Condizione di hold cilindro durante movimento
END_VAR
VAR_OUTPUT
  OUT_EV_Forward : BOOL ;	//Uscita PLC A..
  OUT_EV_Back : BOOL ;	//Uscita PLC A..
  OUT_State_CylForward : BOOL ;	//Stato cilindro avanti
  OUT_State_CylBack : BOOL ;	//Stato cilindro indietro
  OUT_Alarm_ES_Forward : BOOL ;	//Allarme finecorsa avanti
  OUT_Alarm_ES_Back : BOOL ;	//Allarme finecorsa indietro
  OUT_Alarm_ForwBack : BOOL ;	//Allarme corto micro
  OUT_State_CylHold : BOOL ;	//Cilindro in stato di hold
END_VAR
VAR
  FP_IN_Comando_Avanti : BOOL ;
  FP_IN_Comando_Indietro : BOOL ;
  FP_ResetAllarmi : BOOL ;
  Timer1 : SFB 4;
  Timer2 : SFB 4;
END_VAR
VAR_TEMP
  Timer1_IN : BOOL ;
  Timer1_OUT : BOOL ;
  Timer2_IN : BOOL ;
  Timer2_OUT : BOOL ;
END_VAR
BEGIN
NETWORK
TITLE = FUNZIONE CILINDRO
//START CASE
// CASE: OFF
// CASE: ON
// CASE: DIS
//END CASE
//STATES
//HOLD
//ALARMS RESET
// ALLARM ON
// ALLARM OFF
// ALLARM ON OFF
NETWORK
TITLE =
      A     #IN_Alarms_Reset;
      A(;
      A     #IN_EndStroke_Forward;
      O     #IN_EndStroke_Back;
      );
      R     #OUT_State_CylHold;
NETWORK
TITLE = Select Case
//Condizioni per uscite elettrovalvole
      A     #IN_Command_CylForward;
      FP    #FP_IN_Comando_Avanti;
      O(;
      A     #IN_Command_CylBack;
      FP    #FP_IN_Comando_Indietro;
      );
      AN    #IN_Hold_Condition;
      R     #OUT_State_CylHold;
      AN    #IN_Enable;
      O     #OUT_State_CylHold;
      JC    DIS;
//-
      A     #IN_Command_CylForward;
      AN    #IN_Hold_Condition;
      JC    AV;
//-
      A     #IN_Command_CylBack;
      AN    #IN_Hold_Condition;
      JC    IND;
//-
      JU    ENDC;
NETWORK
TITLE = CASE: OFF
// Cilindro comandato in posizione "riposo"
IND:  NOP   0;
      SET;
      S     #OUT_EV_Back;
      R     #OUT_EV_Forward;
      JU    ENDC;
NETWORK
TITLE = CASE: ON
// Cilindro comandato in posizione "attivo"
AV:   NOP   0;
      SET;
      R     #OUT_EV_Back;
      S     #OUT_EV_Forward;
      JU    ENDC;
NETWORK
TITLE = CASE: DISABLE
// Uscite disabilitate
DIS:  NOP   0;
      SET;
      R     #OUT_EV_Back;
      R     #OUT_EV_Forward;
NETWORK
TITLE = END CASE
ENDC: NOP   0;
NETWORK
TITLE = STATES
// Cilindro in posizione "attivo"
      A     #IN_EndStroke_Forward;
      AN    #IN_EndStroke_Back;
      AN    #OUT_State_CylHold;
      =     #OUT_State_CylForward;
// Cilindro in posizione "riposo"
      AN    #IN_EndStroke_Forward;
      A     #IN_EndStroke_Back;
      AN    #OUT_State_CylHold;
      =     #OUT_State_CylBack;
NETWORK
TITLE = HOLD
// Abilita hold se barriera durante movimento
      A(;
      A     #OUT_EV_Forward;
      AN    #OUT_State_CylForward;
      A     #IN_Hold_Condition;
      O;
      A     #OUT_EV_Back;
      AN    #OUT_State_CylBack;
      A     #IN_Hold_Condition;
      );
      A     #IN_Enable;
      S     #OUT_State_CylHold;
NETWORK
TITLE = ALARMS RESET
// Reset allarmi
      A     #IN_Alarms_Reset;
      FP    #FP_ResetAllarmi;
      R     #OUT_Alarm_ES_Forward;
      R     #OUT_Alarm_ES_Back;
      R     #OUT_Alarm_ForwBack;
NETWORK
TITLE = Allarme Cilindro avanti non segnalato
// Cilindro non spostato in posizione "attivo" in tempo utile
      A     #OUT_EV_Forward;
      AN    #OUT_State_CylForward;
      AN    #IN_Hold_Condition;
      A     #IN_Enable;
      =     #Timer1_IN;
      BLD   16;
      =     L 7.0;
      L     DINO;
      T     LW 5;
      CDB;
      OPN   DI [LW 5];
      TAR2  LD 1;
      A     #Timer1_IN;
      =     DIX [AR2,P#12.0];
      L     DBD [AR2,P#2.0];
      T     DID [AR2,P#14.0];
      +AR2  P#12.0;
      UC    SFB 4;
      LAR2  LD 1;
      A     DIX [AR2,P#18.0];
      =     #Timer1_OUT;
      CDB;
      BLD   17;
      A     #Timer1_OUT;
      S     #OUT_Alarm_ES_Forward;
NETWORK
TITLE = Allarme Cilindro indietro non segnalato
// Cilindro non tornato in posizione "riposo" in tempo utile
      A     #OUT_EV_Back;
      AN    #OUT_State_CylBack;
      AN    #IN_Hold_Condition;
      A     #IN_Enable;
      =     #Timer2_IN;
      BLD   16;
      =     L 7.0;
      L     DINO;
      T     LW 5;
      CDB;
      OPN   DI [LW 5];
      TAR2  LD 1;
      A     #Timer2_IN;
      =     DIX [AR2,P#34.0];
      L     DBD [AR2,P#2.0];
      T     DID [AR2,P#36.0];
      +AR2  P#34.0;
      UC    SFB 4;
      LAR2  LD 1;
      A     DIX [AR2,P#40.0];
      =     #Timer2_OUT;
      CDB;
      BLD   17;
      A     #Timer2_OUT;
      S     #OUT_Alarm_ES_Back;
NETWORK
TITLE = Allarme Cilindro avanti e indietro entrambi attivi
// Micro contemporanei
      A     #IN_EndStroke_Forward;
      A     #IN_EndStroke_Back;
      A     #IN_Enable;
      S     #OUT_Alarm_ForwBack;
NETWORK
TITLE = Fine
      NOP   0;
NETWORK
TITLE = ALARMS RESET
// Reset allarmi
      A     #IN_Alarms_Reset;
      FP    #FP_ResetAllarmi;
      R     #OUT_Alarm_ES_Forward;
      R     #OUT_Alarm_ES_Back;
      R     #OUT_Alarm_ForwBack;
END_FUNCTION_BLOCK

